LIN {X 0,Y 416.855,Z 989.857,A -85,B 0,C 180,E1 6681.651,E2 6681.651} C_VEL
LIN {X 0,Y 426.001,Z 970.369,A -85,B 0,C 180,E1 6680.53,E2 6680.53} C_VEL
LIN {X 0,Y 436.146,Z 946.367,A -85,B 0,C 180,E1 6679.376,E2 6679.376} C_VEL
LIN {X 0,Y 445.2,Z 921.165,A -85,B 0,C 180,E1 6678.399,E2 6678.399} C_VEL
LIN {X 0,Y 451.671,Z 900.478,A -85,B 0,C 180,E1 6677.741,E2 6677.741} C_VEL
LIN {X 0,Y 457.353,Z 879.296,A -85,B 0,C 180,E1 6677.183,E2 6677.183} C_VEL
LIN {X 0,Y 462.4,Z 856.717,A -85,B 0,C 180,E1 6676.706,E2 6676.706} C_VEL
LIN {X 0,Y 467.347,Z 827.03,A -85,B 0,C 180,E1 6676.196,E2 6676.196} C_VEL
LIN {X 0,Y 472.981,Z 773.128,A -85,B 0,C 180,E1 6675.392,E2 6675.392} C_VEL
LIN {X 0,Y 490.265,Z 601.502,A -85,B 0,C 180,E1 6672.888,E2 6672.888} C_VEL
LIN {X 0,Y 487.784,Z 596.947,A -85,B 0,C 180,E1 6670.631,E2 6670.631} C_VEL
LIN {X 0,Y 485.782,Z 593.042,A -85,B 0,C 180,E1 6668.101,E2 6668.101} C_VEL
LIN {X 0,Y 484.292,Z 588.607,A -85,B 0,C 180,E1 6662.84,E2 6662.84} C_VEL
LIN {X 0,Y 486.143,Z 593.645,A -85,B 0,C 180,E1 6657.171,E2 6657.171} C_VEL
LIN {X 0,Y 488.529,Z 598.315,A -85,B 0,C 180,E1 6654.421,E2 6654.421} C_VEL
LIN {X 0,Y 490.215,Z 601.519,A -85,B 0,C 180,E1 6652.939,E2 6652.939} C_VEL
LIN {X 0,Y 468.422,Z 816.947,A -85,B 0,C 180,E1 6649.795,E2 6649.795} C_VEL
LIN {X 0,Y 465.267,Z 839.316,A -85,B 0,C 180,E1 6649.432,E2 6649.432} C_VEL
LIN {X 0,Y 460.997,Z 861.82,A -85,B 0,C 180,E1 6649.009,E2 6649.009} C_VEL
LIN {X 0,Y 454.539,Z 888.776,A -85,B 0,C 180,E1 6648.359,E2 6648.359} C_VEL
LIN {X 0,Y 447.193,Z 913.264,A -85,B 0,C 180,E1 6647.605,E2 6647.605} C_VEL
LIN {X 0,Y 440.015,Z 933.977,A -85,B 0,C 180,E1 6646.83,E2 6646.83} C_VEL
LIN {X 0,Y 432.19,Z 953.973,A -85,B 0,C 180,E1 6645.941,E2 6645.941} C_VEL
LIN {X 0,Y 422.719,Z 975.589,A -85,B 0,C 180,E1 6644.807,E2 6644.807} C_VEL
LIN {X 0,Y 410.412,Z 1000.373,A -85,B 0,C 180,E1 6643.224,E2 6643.224} C_VEL
LIN {X 0,Y 400.027,Z 1019.259,A -85,B 0,C 180,E1 6641.769,E2 6641.769} C_VEL
LIN {X 0,Y 389.898,Z 1036.281,A -85,B 0,C 180,E1 6640.244,E2 6640.244} C_VEL
LIN {X 0,Y 379.202,Z 1053.022,A -85,B 0,C 180,E1 6638.499,E2 6638.499} C_VEL
LIN {X 0,Y 365.53,Z 1073.081,A -85,B 0,C 180,E1 6636.01,E2 6636.01} C_VEL
LIN {X 0,Y 351.999,Z 1091.305,A -85,B 0,C 180,E1 6633.222,E2 6633.222} C_VEL
LIN {X 0,Y 340.838,Z 1105.652,A -85,B 0,C 180,E1 6630.605,E2 6630.605} C_VEL
LIN {X 0,Y 329.999,Z 1119.088,A -85,B 0,C 180,E1 6627.708,E2 6627.708} C_VEL
LIN {X 0,Y 317.403,Z 1134.331,A -85,B 0,C 180,E1 6623.749,E2 6623.749} C_VEL
LIN {X 0,Y 306.251,Z 1147.367,A -85,B 0,C 180,E1 6619.526,E2 6619.526} C_VEL
LIN {X 0,Y 297.848,Z 1157.309,A -85,B 0,C 180,E1 6615.645,E2 6615.645} C_VEL
LIN {X 0,Y 290.31,Z 1166.501,A -85,B 0,C 180,E1 6611.336,E2 6611.336} C_VEL
LIN {X 0,Y 282.575,Z 1176.52,A -85,B 0,C 180,E1 6605.471,E2 6605.471} C_VEL
LIN {X 0,Y 278.125,Z 1182.904,A -85,B 0,C 180,E1 6600.696,E2 6600.696} C_VEL
LIN {X 0,Y 275.171,Z 1187.842,A -85,B 0,C 180,E1 6596.082,E2 6596.082} C_VEL
LIN {X 0,Y 273.379,Z 1191.521,A -85,B 0,C 180,E1 6591.678,E2 6591.678} C_VEL
LIN {X 0,Y 272.422,Z 1194.229,A -85,B 0,C 180,E1 6587.294,E2 6587.294} C_VEL
LIN {X 0,Y 272.031,Z 1195.927,A -85,B 0,C 180,E1 6583.172,E2 6583.172} C_VEL
LIN {X 0,Y 271.932,Z 1196.773,A -85,B 0,C 180,E1 6579.31,E2 6579.31} C_VEL
LIN {X 0,Y 271.908,Z 1196.87,A -85,B 0,C 180,E1 6575.274,E2 6575.274} C_VEL
LIN {X 0,Y 271.941,Z 1196.163,A -85,B 0,C 180,E1 6571.263,E2 6571.263} C_VEL
LIN {X 0,Y 272.119,Z 1194.546,A -85,B 0,C 180,E1 6567.05,E2 6567.05} C_VEL
LIN {X 0,Y 272.714,Z 1191.882,A -85,B 0,C 180,E1 6562.626,E2 6562.626} C_VEL
LIN {X 0,Y 273.987,Z 1188.224,A -85,B 0,C 180,E1 6558.207,E2 6558.207} C_VEL
LIN {X 0,Y 276.136,Z 1183.547,A -85,B 0,C 180,E1 6553.81,E2 6553.81} C_VEL
LIN {X 0,Y 279.466,Z 1177.53,A -85,B 0,C 180,E1 6549.255,E2 6549.255} C_VEL
LIN {X 0,Y 284.504,Z 1169.638,A -85,B 0,C 180,E1 6544.387,E2 6544.387} C_VEL
LIN {X 0,Y 291.973,Z 1158.86,A -85,B 0,C 180,E1 6539.09,E2 6539.09} C_VEL
LIN {X 0,Y 299.509,Z 1148.546,A -85,B 0,C 180,E1 6534.956,E2 6534.956} C_VEL
LIN {X 0,Y 307.424,Z 1137.911,A -85,B 0,C 180,E1 6531.356,E2 6531.356} C_VEL
LIN {X 0,Y 316.822,Z 1125.344,A -85,B 0,C 180,E1 6527.761,E2 6527.761} C_VEL
LIN {X 0,Y 329.366,Z 1108.186,A -85,B 0,C 180,E1 6523.737,E2 6523.737} C_VEL
LIN {X 0,Y 339.219,Z 1094.184,A -85,B 0,C 180,E1 6521.01,E2 6521.01} C_VEL
LIN {X 0,Y 349.142,Z 1079.549,A -85,B 0,C 180,E1 6518.572,E2 6518.572} C_VEL
LIN {X 0,Y 359.626,Z 1063.349,A -85,B 0,C 180,E1 6516.264,E2 6516.264} C_VEL
LIN {X 0,Y 372.238,Z 1042.639,A -85,B 0,C 180,E1 6513.782,E2 6513.782} C_VEL
LIN {X 0,Y 383.807,Z 1021.754,A -85,B 0,C 180,E1 6511.724,E2 6511.724} C_VEL
LIN {X 0,Y 393.285,Z 1003.316,A -85,B 0,C 180,E1 6510.184,E2 6510.184} C_VEL
LIN {X 0,Y 401.929,Z 985.07,A -85,B 0,C 180,E1 6508.875,E2 6508.875} C_VEL
LIN {X 0,Y 412.234,Z 961.113,A -85,B 0,C 180,E1 6507.409,E2 6507.409} C_VEL
LIN {X 0,Y 421.376,Z 936.508,A -85,B 0,C 180,E1 6506.191,E2 6506.191} C_VEL
LIN {X 0,Y 428.141,Z 915.89,A -85,B 0,C 180,E1 6505.338,E2 6505.338} C_VEL
LIN {X 0,Y 434.12,Z 895.023,A -85,B 0,C 180,E1 6504.612,E2 6504.612} C_VEL
LIN {X 0,Y 434.611,Z 893.203,A -85,B 0,C 180,E1 6504.555,E2 6504.555} C_VEL
LIN {X 0,Y 436.165,Z 886.037,A -85,B 0,C 180,E1 6504.214,E2 6504.214} C_VEL
LIN {X 0,Y 438.207,Z 868.294,A -85,B 0,C 180,E1 6502.999,E2 6502.999} C_VEL
LIN {X 0,Y 439.312,Z 860.964,A -85,B 0,C 180,E1 6502.707,E2 6502.707} C_VEL
LIN {X 0,Y 443.317,Z 838.651,A -85,B 0,C 180,E1 6502.264,E2 6502.264} C_VEL
LIN {X 0,Y 446.283,Z 816.191,A -85,B 0,C 180,E1 6501.884,E2 6501.884} C_VEL
LIN {X 0,Y 466.557,Z 598.28,A -85,B 0,C 180,E1 6498.618,E2 6498.618} C_VEL
LIN {X 0,Y 467.039,Z 592.534,A -85,B 0,C 180,E1 6498.505,E2 6498.505} C_VEL
LIN {X 0,Y 462.723,Z 584.65,A -85,B 0,C 180,E1 6495.864,E2 6495.864} C_VEL
LIN {X 0,Y 459.733,Z 579.467,A -85,B 0,C 180,E1 6493.65,E2 6493.65} C_VEL
LIN {X 0,Y 457.995,Z 576.374,A -85,B 0,C 180,E1 6492.098,E2 6492.098} C_VEL
LIN {X 0,Y 455.895,Z 572.558,A -85,B 0,C 180,E1 6489.723,E2 6489.723} C_VEL
LIN {X 0,Y 453.963,Z 568.532,A -85,B 0,C 180,E1 6486.069,E2 6486.069} C_VEL
LIN {X 0,Y 453.614,Z 568.037,A -85,B 0,C 180,E1 6484.805,E2 6484.805} C_VEL
LIN {X 0,Y 453.911,Z 568.255,A -85,B 0,C 180,E1 6480.252,E2 6480.252} C_VEL
LIN {X 0,Y 455.529,Z 572.159,A -85,B 0,C 180,E1 6476.854,E2 6476.854} C_VEL
LIN {X 0,Y 456.46,Z 573.573,A -85,B 0,C 180,E1 6475.666,E2 6475.666} C_VEL
LIN {X 0,Y 459.168,Z 578.446,A -85,B 0,C 180,E1 6472.933,E2 6472.933} C_VEL
LIN {X 0,Y 461.582,Z 582.786,A -85,B 0,C 180,E1 6471.027,E2 6471.027} C_VEL
LIN {X 0,Y 465.2,Z 589.229,A -85,B 0,C 180,E1 6468.658,E2 6468.658} C_VEL
LIN {X 0,Y 467.122,Z 592.997,A -85,B 0,C 180,E1 6467.535,E2 6467.535} C_VEL
LIN {X 0,Y 446.738,Z 813.471,A -85,B 0,C 180,E1 6464.235,E2 6464.235} C_VEL
LIN {X 0,Y 443.482,Z 839.489,A -85,B 0,C 180,E1 6463.8,E2 6463.8} C_VEL
LIN {X 0,Y 439.573,Z 861.723,A -85,B 0,C 180,E1 6463.373,E2 6463.373} C_VEL
LIN {X 0,Y 434.754,Z 883.632,A -85,B 0,C 180,E1 6462.854,E2 6462.854} C_VEL
LIN {X 0,Y 427.738,Z 910.07,A -85,B 0,C 180,E1 6462.065,E2 6462.065} C_VEL
LIN {X 0,Y 419.555,Z 935.282,A -85,B 0,C 180,E1 6461.108,E2 6461.108} C_VEL
LIN {X 0,Y 412.311,Z 954.975,A -85,B 0,C 180,E1 6460.208,E2 6460.208} C_VEL
LIN {X 0,Y 404.389,Z 974.343,A -85,B 0,C 180,E1 6459.169,E2 6459.169} C_VEL
LIN {X 0,Y 395.523,Z 994.037,A -85,B 0,C 180,E1 6457.928,E2 6457.928} C_VEL
LIN {X 0,Y 383.724,Z 1017.725,A -85,B 0,C 180,E1 6456.151,E2 6456.151} C_VEL
LIN {X 0,Y 372.705,Z 1037.638,A -85,B 0,C 180,E1 6454.345,E2 6454.345} C_VEL
LIN {X 0,Y 362.414,Z 1054.953,A -85,B 0,C 180,E1 6452.499,E2 6452.499} C_VEL
LIN {X 0,Y 351.852,Z 1071.672,A -85,B 0,C 180,E1 6450.41,E2 6450.41} C_VEL
LIN {X 0,Y 338.858,Z 1091.127,A -85,B 0,C 180,E1 6447.518,E2 6447.518} C_VEL
LIN {X 0,Y 326.855,Z 1107.895,A -85,B 0,C 180,E1 6444.462,E2 6444.462} C_VEL
LIN {X 0,Y 316.79,Z 1121.525,A -85,B 0,C 180,E1 6441.514,E2 6441.514} C_VEL
LIN {X 0,Y 307.034,Z 1134.431,A -85,B 0,C 180,E1 6438.225,E2 6438.225} C_VEL
LIN {X 0,Y 296.536,Z 1148.302,A -85,B 0,C 180,E1 6433.996,E2 6433.996} C_VEL
LIN {X 0,Y 287.11,Z 1160.609,A -85,B 0,C 180,E1 6429.334,E2 6429.334} C_VEL
LIN {X 0,Y 280.577,Z 1169.55,A -85,B 0,C 180,E1 6425.262,E2 6425.262} C_VEL
LIN {X 0,Y 275.039,Z 1177.571,A -85,B 0,C 180,E1 6420.91,E2 6420.91} C_VEL
LIN {X 0,Y 270.647,Z 1184.594,A -85,B 0,C 180,E1 6416.317,E2 6416.317} C_VEL
LIN {X 0,Y 266.919,Z 1191.693,A -85,B 0,C 180,E1 6410.525,E2 6410.525} C_VEL
LIN {X 0,Y 264.96,Z 1196.582,A -85,B 0,C 180,E1 6405.094,E2 6405.094} C_VEL
LIN {X 0,Y 264.183,Z 1199.646,A -85,B 0,C 180,E1 6400.468,E2 6400.468} C_VEL
LIN {X 0,Y 263.954,Z 1201.529,A -85,B 0,C 180,E1 6396.308,E2 6396.308} C_VEL
LIN {X 0,Y 263.915,Z 1202.571,A -85,B 0,C 180,E1 6392.172,E2 6392.172} C_VEL
LIN {X 0,Y 263.913,Z 1202.76,A -85,B 0,C 180,E1 6387.83,E2 6387.83} C_VEL
LIN {X 0,Y 263.958,Z 1202.033,A -85,B 0,C 180,E1 6383.476,E2 6383.476} C_VEL
LIN {X 0,Y 264.264,Z 1200.282,A -85,B 0,C 180,E1 6378.875,E2 6378.875} C_VEL
LIN {X 0,Y 265.179,Z 1197.53,A -85,B 0,C 180,E1 6374.248,E2 6374.248} C_VEL
LIN {X 0,Y 266.953,Z 1193.765,A -85,B 0,C 180,E1 6369.616,E2 6369.616} C_VEL
LIN {X 0,Y 269.817,Z 1188.967,A -85,B 0,C 180,E1 6365.011,E2 6365.011} C_VEL
LIN {X 0,Y 274.125,Z 1182.778,A -85,B 0,C 180,E1 6360.242,E2 6360.242} C_VEL
LIN {X 0,Y 280.711,Z 1174.386,A -85,B 0,C 180,E1 6355.008,E2 6355.008} C_VEL
LIN {X 0,Y 289.919,Z 1163.295,A -85,B 0,C 180,E1 6349.582,E2 6349.582} C_VEL
LIN {X 0,Y 298.594,Z 1153.259,A -85,B 0,C 180,E1 6345.585,E2 6345.585} C_VEL
LIN {X 0,Y 308.005,Z 1142.435,A -85,B 0,C 180,E1 6341.971,E2 6341.971} C_VEL
LIN {X 0,Y 319.554,Z 1129.067,A -85,B 0,C 180,E1 6338.246,E2 6338.246} C_VEL
LIN {X 0,Y 333.497,Z 1112.298,A -85,B 0,C 180,E1 6334.464,E2 6334.464} C_VEL
LIN {X 0,Y 345.466,Z 1097.29,A -85,B 0,C 180,E1 6331.69,E2 6331.69} C_VEL
LIN {X 0,Y 356.816,Z 1082.405,A -85,B 0,C 180,E1 6329.367,E2 6329.367} C_VEL
LIN {X 0,Y 369.062,Z 1065.458,A -85,B 0,C 180,E1 6327.13,E2 6327.13} C_VEL
LIN {X 0,Y 384.064,Z 1042.943,A -85,B 0,C 180,E1 6324.691,E2 6324.691} C_VEL
LIN {X 0,Y 394.923,Z 1025.236,A -85,B 0,C 180,E1 6323.106,E2 6323.106} C_VEL
LIN {X 0,Y 405.046,Z 1007.376,A -85,B 0,C 180,E1 6321.733,E2 6321.733} C_VEL
LIN {X 0,Y 414.747,Z 988.785,A -85,B 0,C 180,E1 6320.514,E2 6320.514} C_VEL
LIN {X 0,Y 424.44,Z 968.395,A -85,B 0,C 180,E1 6319.378,E2 6319.378} C_VEL
LIN {X 0,Y 435.63,Z 941.619,A -85,B 0,C 180,E1 6318.155,E2 6318.155} C_VEL
LIN {X 0,Y 443.597,Z 919.527,A -85,B 0,C 180,E1 6317.338,E2 6317.338} C_VEL
LIN {X 0,Y 449.955,Z 899.331,A -85,B 0,C 180,E1 6316.716,E2 6316.716} C_VEL
LIN {X 0,Y 455.67,Z 878.172,A -85,B 0,C 180,E1 6316.176,E2 6316.176} C_VEL
LIN {X 0,Y 461.272,Z 853.11,A -85,B 0,C 180,E1 6315.67,E2 6315.67} C_VEL
LIN {X 0,Y 465.812,Z 824.74,A -85,B 0,C 180,E1 6315.2,E2 6315.2} C_VEL
LIN {X 0,Y 473.898,Z 747.238,A -85,B 0,C 180,E1 6314.062,E2 6314.062} C_VEL
LIN {X 0,Y 488.256,Z 607.87,A -85,B 0,C 180,E1 6312.057,E2 6312.057} C_VEL
LIN {X 0,Y 486.579,Z 604.671,A -85,B 0,C 180,E1 6310.418,E2 6310.418} C_VEL
LIN {X 0,Y 484.772,Z 600.976,A -85,B 0,C 180,E1 6308.063,E2 6308.063} C_VEL
LIN {X 0,Y 483.312,Z 596.579,A -85,B 0,C 180,E1 6302.846,E2 6302.846} C_VEL
LIN {X 0,Y 485.071,Z 601.541,A -85,B 0,C 180,E1 6297.283,E2 6297.283} C_VEL
LIN {X 0,Y 487.35,Z 606.118,A -85,B 0,C 180,E1 6294.584,E2 6294.584} C_VEL
LIN {X 0,Y 488.188,Z 608.003,A -85,B 0,C 180,E1 6293.774,E2 6293.774} C_VEL
LIN {X 0,Y 466.314,Z 819.614,A -85,B 0,C 180,E1 6290.714,E2 6290.714} C_VEL
LIN {X 0,Y 462.847,Z 842.858,A -85,B 0,C 180,E1 6290.338,E2 6290.338} C_VEL
LIN {X 0,Y 456.918,Z 871.614,A -85,B 0,C 180,E1 6289.772,E2 6289.772} C_VEL
LIN {X 0,Y 450.694,Z 895.154,A -85,B 0,C 180,E1 6289.169,E2 6289.169} C_VEL
LIN {X 0,Y 444.315,Z 915.662,A -85,B 0,C 180,E1 6288.53,E2 6288.53} C_VEL
LIN {X 0,Y 437.322,Z 935.333,A -85,B 0,C 180,E1 6287.798,E2 6287.798} C_VEL
LIN {X 0,Y 429.119,Z 955.802,A -85,B 0,C 180,E1 6286.895,E2 6286.895} C_VEL
LIN {X 0,Y 417.977,Z 980.398,A -85,B 0,C 180,E1 6285.594,E2 6285.594} C_VEL
LIN {X 0,Y 406.456,Z 1002.68,A -85,B 0,C 180,E1 6284.153,E2 6284.153} C_VEL
LIN {X 0,Y 396.249,Z 1020.763,A -85,B 0,C 180,E1 6282.761,E2 6282.761} C_VEL
LIN {X 0,Y 386,Z 1037.532,A -85,B 0,C 180,E1 6281.264,E2 6281.264} C_VEL
LIN {X 0,Y 373.867,Z 1056.004,A -85,B 0,C 180,E1 6279.327,E2 6279.327} C_VEL
LIN {X 0,Y 359.225,Z 1076.511,A -85,B 0,C 180,E1 6276.71,E2 6276.71} C_VEL
LIN {X 0,Y 347.305,Z 1092.092,A -85,B 0,C 180,E1 6274.303,E2 6274.303} C_VEL
LIN {X 0,Y 336.022,Z 1106.146,A -85,B 0,C 180,E1 6271.735,E2 6271.735} C_VEL
LIN {X 0,Y 324.838,Z 1119.541,A -85,B 0,C 180,E1 6268.836,E2 6268.836} C_VEL
LIN {X 0,Y 311.789,Z 1134.715,A -85,B 0,C 180,E1 6264.86,E2 6264.86} C_VEL
LIN {X 0,Y 300.671,Z 1147.194,A -85,B 0,C 180,E1 6260.789,E2 6260.789} C_VEL
LIN {X 0,Y 291.825,Z 1157.164,A -85,B 0,C 180,E1 6256.868,E2 6256.868} C_VEL
LIN {X 0,Y 284.076,Z 1166.104,A -85,B 0,C 180,E1 6252.639,E2 6252.639} C_VEL
LIN {X 0,Y 276.368,Z 1175.533,A -85,B 0,C 180,E1 6247.17,E2 6247.17} C_VEL
LIN {X 0,Y 270.789,Z 1182.864,A -85,B 0,C 180,E1 6241.622,E2 6241.622} C_VEL
LIN {X 0,Y 267.559,Z 1187.826,A -85,B 0,C 180,E1 6236.883,E2 6236.883} C_VEL
LIN {X 0,Y 265.582,Z 1191.529,A -85,B 0,C 180,E1 6232.348,E2 6232.348} C_VEL
LIN {X 0,Y 264.503,Z 1194.261,A -85,B 0,C 180,E1 6227.829,E2 6227.829} C_VEL
LIN {X 0,Y 264.055,Z 1195.982,A -85,B 0,C 180,E1 6223.577,E2 6223.577} C_VEL
LIN {X 0,Y 263.934,Z 1196.85,A -85,B 0,C 180,E1 6219.594,E2 6219.594} C_VEL
LIN {X 0,Y 263.909,Z 1196.969,A -85,B 0,C 180,E1 6215.434,E2 6215.434} C_VEL
LIN {X 0,Y 263.941,Z 1196.285,A -85,B 0,C 180,E1 6211.302,E2 6211.302} C_VEL
LIN {X 0,Y 264.144,Z 1194.579,A -85,B 0,C 180,E1 6206.744,E2 6206.744} C_VEL
LIN {X 0,Y 264.803,Z 1191.893,A -85,B 0,C 180,E1 6202.187,E2 6202.187} C_VEL
LIN {X 0,Y 266.209,Z 1188.155,A -85,B 0,C 180,E1 6197.574,E2 6197.574} C_VEL
LIN {X 0,Y 268.513,Z 1183.515,A -85,B 0,C 180,E1 6193.114,E2 6193.114} C_VEL
LIN {X 0,Y 271.894,Z 1177.77,A -85,B 0,C 180,E1 6188.649,E2 6188.649} C_VEL
LIN {X 0,Y 276.938,Z 1170.247,A -85,B 0,C 180,E1 6183.865,E2 6183.865} C_VEL
LIN {X 0,Y 285.017,Z 1159.177,A -85,B 0,C 180,E1 6178.249,E2 6178.249} C_VEL
LIN {X 0,Y 292.974,Z 1148.744,A -85,B 0,C 180,E1 6173.985,E2 6173.985} C_VEL
LIN {X 0,Y 301.094,Z 1138.281,A -85,B 0,C 180,E1 6170.386,E2 6170.386} C_VEL
LIN {X 0,Y 310.348,Z 1126.364,A -85,B 0,C 180,E1 6166.919,E2 6166.919} C_VEL
LIN {X 0,Y 323.031,Z 1109.711,A -85,B 0,C 180,E1 6162.92,E2 6162.92} C_VEL
LIN {X 0,Y 333.957,Z 1094.677,A -85,B 0,C 180,E1 6159.961,E2 6159.961} C_VEL
LIN {X 0,Y 344.155,Z 1080.078,A -85,B 0,C 180,E1 6157.519,E2 6157.519} C_VEL
LIN {X 0,Y 354.584,Z 1064.41,A -85,B 0,C 180,E1 6155.278,E2 6155.278} C_VEL
LIN {X 0,Y 366.856,Z 1044.878,A -85,B 0,C 180,E1 6152.916,E2 6152.916} C_VEL
LIN {X 0,Y 379.299,Z 1023.117,A -85,B 0,C 180,E1 6150.753,E2 6150.753} C_VEL
LIN {X 0,Y 388.761,Z 1005.204,A -85,B 0,C 180,E1 6149.254,E2 6149.254} C_VEL
LIN {X 0,Y 397.394,Z 987.488,A -85,B 0,C 180,E1 6147.975,E2 6147.975} C_VEL
LIN {X 0,Y 405.934,Z 968.287,A -85,B 0,C 180,E1 6146.776,E2 6146.776} C_VEL
LIN {X 0,Y 415.123,Z 945.419,A -85,B 0,C 180,E1 6145.573,E2 6145.573} C_VEL
LIN {X 0,Y 424.04,Z 919.652,A -85,B 0,C 180,E1 6144.469,E2 6144.469} C_VEL
LIN {X 0,Y 430.538,Z 897.744,A -85,B 0,C 180,E1 6143.7,E2 6143.7} C_VEL
LIN {X 0,Y 435.93,Z 876.487,A -85,B 0,C 180,E1 6143.083,E2 6143.083} C_VEL
LIN {X 0,Y 439.312,Z 860.964,A -85,B 0,C 180,E1 6142.707,E2 6142.707} C_VEL
LIN {X 0,Y 440.435,Z 853.582,A -85,B 0,C 180,E1 6142.424,E2 6142.424} C_VEL
LIN {X 0,Y 441.852,Z 834.293,A -85,B 0,C 180,E1 6141.283,E2 6141.283} C_VEL
LIN {X 0,Y 442.463,Z 827.846,A -85,B 0,C 180,E1 6141.087,E2 6141.087} C_VEL
LIN {X 0,Y 447.025,Z 782.963,A -85,B 0,C 180,E1 6140.397,E2 6140.397} C_VEL
LIN {X 0,Y 464.486,Z 598.22,A -85,B 0,C 180,E1 6137.654,E2 6137.654} C_VEL
LIN {X 0,Y 460.671,Z 591.177,A -85,B 0,C 180,E1 6135.162,E2 6135.162} C_VEL
LIN {X 0,Y 458.162,Z 586.637,A -85,B 0,C 180,E1 6133.183,E2 6133.183} C_VEL
LIN {X 0,Y 456.632,Z 583.895,A -85,B 0,C 180,E1 6131.75,E2 6131.75} C_VEL
LIN {X 0,Y 454.824,Z 580.443,A -85,B 0,C 180,E1 6129.618,E2 6129.618} C_VEL
LIN {X 0,Y 452.946,Z 576.425,A -85,B 0,C 180,E1 6125.955,E2 6125.955} C_VEL
LIN {X 0,Y 452.565,Z 575.934,A -85,B 0,C 180,E1 6124.435,E2 6124.435} C_VEL
LIN {X 0,Y 452.919,Z 576.315,A -85,B 0,C 180,E1 6120.253,E2 6120.253} C_VEL
LIN {X 0,Y 454.733,Z 580.388,A -85,B 0,C 180,E1 6116.596,E2 6116.596} C_VEL
LIN {X 0,Y 455.558,Z 581.953,A -85,B 0,C 180,E1 6115.531,E2 6115.531} C_VEL
LIN {X 0,Y 457.887,Z 586.121,A -85,B 0,C 180,E1 6113.165,E2 6113.165} C_VEL
LIN {X 0,Y 460.24,Z 590.471,A -85,B 0,C 180,E1 6111.253,E2 6111.253} C_VEL
LIN {X 0,Y 463.779,Z 596.967,A -85,B 0,C 180,E1 6108.874,E2 6108.874} C_VEL
LIN {X 0,Y 464.522,Z 598.688,A -85,B 0,C 180,E1 6108.405,E2 6108.405} C_VEL
LIN {X 0,Y 443.835,Z 817.103,A -85,B 0,C 180,E1 6105.158,E2 6105.158} C_VEL
LIN {X 0,Y 440.777,Z 840.468,A -85,B 0,C 180,E1 6104.768,E2 6104.768} C_VEL
LIN {X 0,Y 436.776,Z 862.653,A -85,B 0,C 180,E1 6104.346,E2 6104.346} C_VEL
LIN {X 0,Y 431.448,Z 886.228,A -85,B 0,C 180,E1 6103.79,E2 6103.79} C_VEL
LIN {X 0,Y 423.603,Z 914.226,A -85,B 0,C 180,E1 6102.935,E2 6102.935} C_VEL
LIN {X 0,Y 416.546,Z 935.471,A -85,B 0,C 180,E1 6102.131,E2 6102.131} C_VEL
LIN {X 0,Y 408.996,Z 955.598,A -85,B 0,C 180,E1 6101.223,E2 6101.223} C_VEL
LIN {X 0,Y 400.625,Z 975.615,A -85,B 0,C 180,E1 6100.158,E2 6100.158} C_VEL
LIN {X 0,Y 389.678,Z 999.236,A -85,B 0,C 180,E1 6098.659,E2 6098.659} C_VEL
LIN {X 0,Y 378.143,Z 1021.212,A -85,B 0,C 180,E1 6096.953,E2 6096.953} C_VEL
LIN {X 0,Y 368.167,Z 1038.749,A -85,B 0,C 180,E1 6095.35,E2 6095.35} C_VEL
LIN {X 0,Y 357.904,Z 1055.574,A -85,B 0,C 180,E1 6093.558,E2 6093.558} C_VEL
LIN {X 0,Y 346.69,Z 1072.843,A -85,B 0,C 180,E1 6091.395,E2 6091.395} C_VEL
LIN {X 0,Y 332.11,Z 1093.801,A -85,B 0,C 180,E1 6088.205,E2 6088.205} C_VEL
LIN {X 0,Y 320.819,Z 1109.09,A -85,B 0,C 180,E1 6085.366,E2 6085.366} C_VEL
LIN {X 0,Y 310.486,Z 1122.603,A -85,B 0,C 180,E1 6082.393,E2 6082.393} C_VEL
LIN {X 0,Y 299.954,Z 1136.051,A -85,B 0,C 180,E1 6078.883,E2 6078.883} C_VEL
LIN {X 0,Y 287.97,Z 1151.074,A -85,B 0,C 180,E1 6074.049,E2 6074.049} C_VEL
LIN {X 0,Y 279.886,Z 1161.288,A -85,B 0,C 180,E1 6070.02,E2 6070.02} C_VEL
LIN {X 0,Y 273.124,Z 1170.142,A -85,B 0,C 180,E1 6065.856,E2 6065.856} C_VEL
LIN {X 0,Y 267.312,Z 1178.185,A -85,B 0,C 180,E1 6061.328,E2 6061.328} C_VEL
LIN {X 0,Y 261.961,Z 1186.53,A -85,B 0,C 180,E1 6055.551,E2 6055.551} C_VEL
LIN {X 0,Y 258.589,Z 1192.715,A -85,B 0,C 180,E1 6049.894,E2 6049.894} C_VEL
LIN {X 0,Y 256.954,Z 1196.766,A -85,B 0,C 180,E1 6045.113,E2 6045.113} C_VEL
LIN {X 0,Y 256.19,Z 1199.635,A -85,B 0,C 180,E1 6040.571,E2 6040.571} C_VEL
LIN {X 0,Y 255.953,Z 1201.488,A -85,B 0,C 180,E1 6036.281,E2 6036.281} C_VEL
LIN {X 0,Y 255.915,Z 1202.499,A -85,B 0,C 180,E1 6032.016,E2 6032.016} C_VEL
LIN {X 0,Y 255.913,Z 1202.679,A -85,B 0,C 180,E1 6027.762,E2 6027.762} C_VEL
LIN {X 0,Y 255.963,Z 1201.967,A -85,B 0,C 180,E1 6023.271,E2 6023.271} C_VEL
LIN {X 0,Y 256.302,Z 1200.231,A -85,B 0,C 180,E1 6018.525,E2 6018.525} C_VEL
LIN {X 0,Y 257.326,Z 1197.452,A -85,B 0,C 180,E1 6013.693,E2 6013.693} C_VEL
LIN {X 0,Y 259.35,Z 1193.539,A -85,B 0,C 180,E1 6008.753,E2 6008.753} C_VEL
LIN {X 0,Y 262.494,Z 1188.709,A -85,B 0,C 180,E1 6004.021,E2 6004.021} C_VEL
LIN {X 0,Y 267.137,Z 1182.515,A -85,B 0,C 180,E1 5999.152,E2 5999.152} C_VEL
LIN {X 0,Y 274.542,Z 1173.717,A -85,B 0,C 180,E1 5993.585,E2 5993.585} C_VEL
LIN {X 0,Y 284.028,Z 1162.882,A -85,B 0,C 180,E1 5988.273,E2 5988.273} C_VEL
LIN {X 0,Y 292.666,Z 1153.357,A -85,B 0,C 180,E1 5984.437,E2 5984.437} C_VEL
LIN {X 0,Y 302.444,Z 1142.572,A -85,B 0,C 180,E1 5980.795,E2 5980.795} C_VEL
LIN {X 0,Y 313.871,Z 1129.843,A -85,B 0,C 180,E1 5977.213,E2 5977.213} C_VEL
LIN {X 0,Y 328.859,Z 1112.496,A -85,B 0,C 180,E1 5973.269,E2 5973.269} C_VEL
LIN {X 0,Y 341.184,Z 1097.521,A -85,B 0,C 180,E1 5970.505,E2 5970.505} C_VEL
LIN {X 0,Y 352.831,Z 1082.673,A -85,B 0,C 180,E1 5968.198,E2 5968.198} C_VEL
LIN {X 0,Y 365.017,Z 1066.252,A -85,B 0,C 180,E1 5966.043,E2 5966.043} C_VEL
LIN {X 0,Y 379.964,Z 1044.518,A -85,B 0,C 180,E1 5963.688,E2 5963.688} C_VEL
LIN {X 0,Y 392.109,Z 1025.138,A -85,B 0,C 180,E1 5961.97,E2 5961.97} C_VEL
LIN {X 0,Y 402.277,Z 1007.566,A -85,B 0,C 180,E1 5960.643,E2 5960.643} C_VEL
LIN {X 0,Y 412.4,Z 988.52,A -85,B 0,C 180,E1 5959.416,E2 5959.416} C_VEL
LIN {X 0,Y 422.721,Z 967.135,A -85,B 0,C 180,E1 5958.256,E2 5958.256} C_VEL
LIN {X 0,Y 433.631,Z 941.281,A -85,B 0,C 180,E1 5957.108,E2 5957.108} C_VEL
LIN {X 0,Y 441.292,Z 920.418,A -85,B 0,C 180,E1 5956.352,E2 5956.352} C_VEL
LIN {X 0,Y 447.952,Z 899.648,A -85,B 0,C 180,E1 5955.723,E2 5955.723} C_VEL
LIN {X 0,Y 453.8,Z 878.354,A -85,B 0,C 180,E1 5955.192,E2 5955.192} C_VEL
LIN {X 0,Y 459.311,Z 854.109,A -85,B 0,C 180,E1 5954.712,E2 5954.712} C_VEL
LIN {X 0,Y 464.11,Z 824.968,A -85,B 0,C 180,E1 5954.235,E2 5954.235} C_VEL
LIN {X 0,Y 471.725,Z 753.59,A -85,B 0,C 180,E1 5953.198,E2 5953.198} C_VEL
LIN {X 0,Y 486.332,Z 614.23,A -85,B 0,C 180,E1 5951.203,E2 5951.203} C_VEL
LIN {X 0,Y 484.867,Z 611.502,A -85,B 0,C 180,E1 5949.616,E2 5949.616} C_VEL
LIN {X 0,Y 483.641,Z 608.779,A -85,B 0,C 180,E1 5947.843,E2 5947.843} C_VEL
LIN {X 0,Y 482.32,Z 604.661,A -85,B 0,C 180,E1 5942.733,E2 5942.733} C_VEL
LIN {X 0,Y 484,Z 609.437,A -85,B 0,C 180,E1 5937.395,E2 5937.395} C_VEL
LIN {X 0,Y 486.175,Z 613.92,A -85,B 0,C 180,E1 5934.749,E2 5934.749} C_VEL
LIN {X 0,Y 486.28,Z 614.379,A -85,B 0,C 180,E1 5934.618,E2 5934.618} C_VEL
LIN {X 0,Y 464.53,Z 820.666,A -85,B 0,C 180,E1 5931.666,E2 5931.666} C_VEL
LIN {X 0,Y 460.616,Z 846.004,A -85,B 0,C 180,E1 5931.26,E2 5931.26} C_VEL
LIN {X 0,Y 454.561,Z 873.901,A -85,B 0,C 180,E1 5930.707,E2 5930.707} C_VEL
LIN {X 0,Y 448.785,Z 895.326,A -85,B 0,C 180,E1 5930.165,E2 5930.165} C_VEL
LIN {X 0,Y 442.293,Z 915.88,A -85,B 0,C 180,E1 5929.538,E2 5929.538} C_VEL
LIN {X 0,Y 435.197,Z 935.532,A -85,B 0,C 180,E1 5928.823,E2 5928.823} C_VEL
LIN {X 0,Y 426.43,Z 957.016,A -85,B 0,C 180,E1 5927.892,E2 5927.892} C_VEL
LIN {X 0,Y 414.347,Z 982.869,A -85,B 0,C 180,E1 5926.528,E2 5926.528} C_VEL
LIN {X 0,Y 403.508,Z 1003.375,A -85,B 0,C 180,E1 5925.212,E2 5925.212} C_VEL
LIN {X 0,Y 393.411,Z 1020.899,A -85,B 0,C 180,E1 5923.883,E2 5923.883} C_VEL
LIN {X 0,Y 382.535,Z 1038.308,A -85,B 0,C 180,E1 5922.35,E2 5922.35} C_VEL
LIN {X 0,Y 368.608,Z 1058.981,A -85,B 0,C 180,E1 5920.179,E2 5920.179} C_VEL
LIN {X 0,Y 354.437,Z 1078.042,A -85,B 0,C 180,E1 5917.711,E2 5917.711} C_VEL
LIN {X 0,Y 342.595,Z 1093.063,A -85,B 0,C 180,E1 5915.383,E2 5915.383} C_VEL
LIN {X 0,Y 330.683,Z 1107.426,A -85,B 0,C 180,E1 5912.741,E2 5912.741} C_VEL
LIN {X 0,Y 316.764,Z 1123.552,A -85,B 0,C 180,E1 5909.155,E2 5909.155} C_VEL
LIN {X 0,Y 304.091,Z 1137.439,A -85,B 0,C 180,E1 5905.286,E2 5905.286} C_VEL
LIN {X 0,Y 294.254,Z 1148.073,A -85,B 0,C 180,E1 5901.714,E2 5901.714} C_VEL
LIN {X 0,Y 285.512,Z 1157.487,A -85,B 0,C 180,E1 5897.938,E2 5897.938} C_VEL
LIN {X 0,Y 277.187,Z 1166.618,A -85,B 0,C 180,E1 5893.525,E2 5893.525} C_VEL
LIN {X 0,Y 268.614,Z 1176.478,A -85,B 0,C 180,E1 5887.545,E2 5887.545} C_VEL
LIN {X 0,Y 263.322,Z 1183.081,A -85,B 0,C 180,E1 5882.37,E2 5882.37} C_VEL
LIN {X 0,Y 259.859,Z 1188.019,A -85,B 0,C 180,E1 5877.498,E2 5877.498} C_VEL
LIN {X 0,Y 257.733,Z 1191.698,A -85,B 0,C 180,E1 5872.826,E2 5872.826} C_VEL
LIN {X 0,Y 256.556,Z 1194.406,A -85,B 0,C 180,E1 5868.166,E2 5868.166} C_VEL
LIN {X 0,Y 256.069,Z 1196.104,A -85,B 0,C 180,E1 5863.779,E2 5863.779} C_VEL
LIN {X 0,Y 255.935,Z 1196.949,A -85,B 0,C 180,E1 5859.67,E2 5859.67} C_VEL
LIN {X 0,Y 255.909,Z 1197.069,A -85,B 0,C 180,E1 5855.605,E2 5855.605} C_VEL
LIN {X 0,Y 255.944,Z 1196.339,A -85,B 0,C 180,E1 5851.118,E2 5851.118} C_VEL
LIN {X 0,Y 256.153,Z 1194.723,A -85,B 0,C 180,E1 5846.642,E2 5846.642} C_VEL
LIN {X 0,Y 256.853,Z 1192.061,A -85,B 0,C 180,E1 5841.943,E2 5841.943} C_VEL
LIN {X 0,Y 258.315,Z 1188.404,A -85,B 0,C 180,E1 5837.253,E2 5837.253} C_VEL
LIN {X 0,Y 260.783,Z 1183.73,A -85,B 0,C 180,E1 5832.598,E2 5832.598} C_VEL
LIN {X 0,Y 264.353,Z 1178.009,A -85,B 0,C 180,E1 5828.009,E2 5828.009} C_VEL
LIN {X 0,Y 269.396,Z 1170.857,A -85,B 0,C 180,E1 5823.313,E2 5823.313} C_VEL
LIN {X 0,Y 277.443,Z 1160.389,A -85,B 0,C 180,E1 5817.765,E2 5817.765} C_VEL
LIN {X 0,Y 286.298,Z 1149.229,A -85,B 0,C 180,E1 5813.079,E2 5813.079} C_VEL
LIN {X 0,Y 294.855,Z 1138.65,A -85,B 0,C 180,E1 5809.376,E2 5809.376} C_VEL
LIN {X 0,Y 304.448,Z 1126.758,A -85,B 0,C 180,E1 5805.872,E2 5805.872} C_VEL
LIN {X 0,Y 317.227,Z 1110.609,A -85,B 0,C 180,E1 5801.938,E2 5801.938} C_VEL
LIN {X 0,Y 329.414,Z 1094.341,A -85,B 0,C 180,E1 5798.731,E2 5798.731} C_VEL
LIN {X 0,Y 339.928,Z 1079.696,A -85,B 0,C 180,E1 5796.297,E2 5796.297} C_VEL
LIN {X 0,Y 350.983,Z 1063.486,A -85,B 0,C 180,E1 5794.003,E2 5794.003} C_VEL
LIN {X 0,Y 364.344,Z 1042.576,A -85,B 0,C 180,E1 5791.533,E2 5791.533} C_VEL
LIN {X 0,Y 376.341,Z 1021.859,A -85,B 0,C 180,E1 5789.527,E2 5789.527} C_VEL
LIN {X 0,Y 386.224,Z 1003.404,A -85,B 0,C 180,E1 5788.017,E2 5788.017} C_VEL
LIN {X 0,Y 395.23,Z 985.139,A -85,B 0,C 180,E1 5786.741,E2 5786.741} C_VEL
LIN {X 0,Y 405.602,Z 961.917,A -85,B 0,C 180,E1 5785.354,E2 5785.354} C_VEL
LIN {X 0,Y 415.289,Z 936.857,A -85,B 0,C 180,E1 5784.145,E2 5784.145} C_VEL
LIN {X 0,Y 422.408,Z 915.858,A -85,B 0,C 180,E1 5783.302,E2 5783.302} C_VEL
LIN {X 0,Y 428.597,Z 894.923,A -85,B 0,C 180,E1 5782.6,E2 5782.6} C_VEL
LIN {X 0,Y 434.571,Z 871.147,A -85,B 0,C 180,E1 5781.947,E2 5781.947} C_VEL
LIN {X 0,Y 440.176,Z 842.487,A -85,B 0,C 180,E1 5781.345,E2 5781.345} C_VEL
LIN {X 0,Y 442.463,Z 827.846,A -85,B 0,C 180,E1 5781.087,E2 5781.087} C_VEL
LIN {X 0,Y 443.043,Z 820.326,A -85,B 0,C 180,E1 5780.847,E2 5780.847} C_VEL
LIN {X 0,Y 443.261,Z 800.783,A -85,B 0,C 180,E1 5779.766,E2 5779.766} C_VEL
LIN {X 0,Y 443.655,Z 794.3,A -85,B 0,C 180,E1 5779.576,E2 5779.576} C_VEL
LIN {X 0,Y 462.005,Z 603.818,A -85,B 0,C 180,E1 5776.771,E2 5776.771} C_VEL
LIN {X 0,Y 458.002,Z 596.246,A -85,B 0,C 180,E1 5773.895,E2 5773.895} C_VEL
LIN {X 0,Y 455.53,Z 591.801,A -85,B 0,C 180,E1 5771.651,E2 5771.651} C_VEL
LIN {X 0,Y 453.755,Z 588.328,A -85,B 0,C 180,E1 5769.513,E2 5769.513} C_VEL
LIN {X 0,Y 451.796,Z 583.984,A -85,B 0,C 180,E1 5765.334,E2 5765.334} C_VEL
LIN {X 0,Y 451.877,Z 584.028,A -85,B 0,C 180,E1 5760.507,E2 5760.507} C_VEL
LIN {X 0,Y 453.563,Z 588.142,A -85,B 0,C 180,E1 5756.841,E2 5756.841} C_VEL
LIN {X 0,Y 454.362,Z 589.632,A -85,B 0,C 180,E1 5755.772,E2 5755.772} C_VEL
LIN {X 0,Y 456.679,Z 593.932,A -85,B 0,C 180,E1 5753.336,E2 5753.336} C_VEL
LIN {X 0,Y 458.906,Z 598.154,A -85,B 0,C 180,E1 5751.48,E2 5751.48} C_VEL
LIN {X 0,Y 462.046,Z 604.17,A -85,B 0,C 180,E1 5749.288,E2 5749.288} C_VEL
LIN {X 0,Y 441.23,Z 819.116,A -85,B 0,C 180,E1 5746.119,E2 5746.119} C_VEL
LIN {X 0,Y 438.196,Z 841.451,A -85,B 0,C 180,E1 5745.748,E2 5745.748} C_VEL
LIN {X 0,Y 434.015,Z 864.023,A -85,B 0,C 180,E1 5745.322,E2 5745.322} C_VEL
LIN {X 0,Y 427.709,Z 890.935,A -85,B 0,C 180,E1 5744.682,E2 5744.682} C_VEL
LIN {X 0,Y 420.415,Z 915.761,A -85,B 0,C 180,E1 5743.913,E2 5743.913} C_VEL
LIN {X 0,Y 413.673,Z 935.657,A -85,B 0,C 180,E1 5743.169,E2 5743.169} C_VEL
LIN {X 0,Y 406.184,Z 955.29,A -85,B 0,C 180,E1 5742.3,E2 5742.3} C_VEL
LIN {X 0,Y 397.982,Z 974.609,A -85,B 0,C 180,E1 5741.293,E2 5741.293} C_VEL
LIN {X 0,Y 388.322,Z 995.222,A -85,B 0,C 180,E1 5740.023,E2 5740.023} C_VEL
LIN {X 0,Y 375.73,Z 1019.243,A -85,B 0,C 180,E1 5738.241,E2 5738.241} C_VEL
LIN {X 0,Y 364.635,Z 1038.383,A -85,B 0,C 180,E1 5736.527,E2 5736.527} C_VEL
LIN {X 0,Y 353.883,Z 1055.62,A -85,B 0,C 180,E1 5734.709,E2 5734.709} C_VEL
LIN {X 0,Y 342.458,Z 1072.787,A -85,B 0,C 180,E1 5732.573,E2 5732.573} C_VEL
LIN {X 0,Y 327.541,Z 1093.651,A -85,B 0,C 180,E1 5729.414,E2 5729.414} C_VEL
LIN {X 0,Y 315.923,Z 1108.916,A -85,B 0,C 180,E1 5726.584,E2 5726.584} C_VEL
LIN {X 0,Y 305.393,Z 1122.248,A -85,B 0,C 180,E1 5723.652,E2 5723.652} C_VEL
LIN {X 0,Y 294.972,Z 1135.07,A -85,B 0,C 180,E1 5720.307,E2 5720.307} C_VEL
LIN {X 0,Y 282.661,Z 1149.986,A -85,B 0,C 180,E1 5715.54,E2 5715.54} C_VEL
LIN {X 0,Y 273.394,Z 1161.128,A -85,B 0,C 180,E1 5711.113,E2 5711.113} C_VEL
LIN {X 0,Y 266.305,Z 1169.948,A -85,B 0,C 180,E1 5706.894,E2 5706.894} C_VEL
LIN {X 0,Y 260.17,Z 1177.992,A -85,B 0,C 180,E1 5702.273,E2 5702.273} C_VEL
LIN {X 0,Y 254.479,Z 1186.349,A -85,B 0,C 180,E1 5696.36,E2 5696.36} C_VEL
LIN {X 0,Y 250.815,Z 1192.611,A -85,B 0,C 180,E1 5690.471,E2 5690.471} C_VEL
LIN {X 0,Y 249.044,Z 1196.687,A -85,B 0,C 180,E1 5685.51,E2 5685.51} C_VEL
LIN {X 0,Y 248.223,Z 1199.509,A -85,B 0,C 180,E1 5680.914,E2 5680.914} C_VEL
LIN {X 0,Y 247.96,Z 1201.377,A -85,B 0,C 180,E1 5676.484,E2 5676.484} C_VEL
LIN {X 0,Y 247.915,Z 1202.404,A -85,B 0,C 180,E1 5672.081,E2 5672.081} C_VEL
LIN {X 0,Y 247.914,Z 1202.599,A -85,B 0,C 180,E1 5667.689,E2 5667.689} C_VEL
LIN {X 0,Y 247.969,Z 1201.901,A -85,B 0,C 180,E1 5663.053,E2 5663.053} C_VEL
LIN {X 0,Y 248.358,Z 1200.129,A -85,B 0,C 180,E1 5658.048,E2 5658.048} C_VEL
LIN {X 0,Y 249.528,Z 1197.298,A -85,B 0,C 180,E1 5652.992,E2 5652.992} C_VEL
LIN {X 0,Y 251.673,Z 1193.52,A -85,B 0,C 180,E1 5648.072,E2 5648.072} C_VEL
LIN {X 0,Y 255.049,Z 1188.708,A -85,B 0,C 180,E1 5643.204,E2 5643.204} C_VEL
LIN {X 0,Y 259.747,Z 1182.835,A -85,B 0,C 180,E1 5638.432,E2 5638.432} C_VEL
LIN {X 0,Y 266.495,Z 1175.161,A -85,B 0,C 180,E1 5633.377,E2 5633.377} C_VEL
LIN {X 0,Y 276.955,Z 1163.903,A -85,B 0,C 180,E1 5627.538,E2 5627.538} C_VEL
LIN {X 0,Y 286.85,Z 1153.456,A -85,B 0,C 180,E1 5623.239,E2 5623.239} C_VEL
LIN {X 0,Y 297.378,Z 1142.332,A -85,B 0,C 180,E1 5619.456,E2 5619.456} C_VEL
LIN {X 0,Y 310.072,Z 1128.733,A -85,B 0,C 180,E1 5615.649,E2 5615.649} C_VEL
LIN {X 0,Y 325.023,Z 1111.937,A -85,B 0,C 180,E1 5611.891,E2 5611.891} C_VEL
LIN {X 0,Y 337.055,Z 1097.752,A -85,B 0,C 180,E1 5609.292,E2 5609.292} C_VEL
LIN {X 0,Y 349.005,Z 1082.937,A -85,B 0,C 180,E1 5607.003,E2 5607.003} C_VEL
LIN {X 0,Y 361.58,Z 1066.42,A -85,B 0,C 180,E1 5604.856,E2 5604.856} C_VEL
LIN {X 0,Y 376.755,Z 1044.894,A -85,B 0,C 180,E1 5602.549,E2 5602.549} C_VEL
LIN {X 0,Y 389.391,Z 1025.148,A -85,B 0,C 180,E1 5600.826,E2 5600.826} C_VEL
LIN {X 0,Y 399.906,Z 1007.319,A -85,B 0,C 180,E1 5599.509,E2 5599.509} C_VEL
LIN {X 0,Y 410.206,Z 988.257,A -85,B 0,C 180,E1 5598.306,E2 5598.306} C_VEL
LIN {X 0,Y 421.236,Z 965.733,A -85,B 0,C 180,E1 5597.118,E2 5597.118} C_VEL
LIN {X 0,Y 431.78,Z 940.953,A -85,B 0,C 180,E1 5596.053,E2 5596.053} C_VEL
LIN {X 0,Y 439.553,Z 920.059,A -85,B 0,C 180,E1 5595.316,E2 5595.316} C_VEL
LIN {X 0,Y 446.304,Z 899.246,A -85,B 0,C 180,E1 5594.702,E2 5594.702} C_VEL
LIN {X 0,Y 452.265,Z 877.766,A -85,B 0,C 180,E1 5594.184,E2 5594.184} C_VEL
LIN {X 0,Y 458.229,Z 851.652,A -85,B 0,C 180,E1 5593.685,E2 5593.685} C_VEL
LIN {X 0,Y 462.719,Z 823.788,A -85,B 0,C 180,E1 5593.242,E2 5593.242} C_VEL
LIN {X 0,Y 473.756,Z 721.234,A -85,B 0,C 180,E1 5591.778,E2 5591.778} C_VEL
LIN {X 0,Y 484.514,Z 620.622,A -85,B 0,C 180,E1 5590.343,E2 5590.343} C_VEL
LIN {X 0,Y 482.592,Z 616.667,A -85,B 0,C 180,E1 5587.74,E2 5587.74} C_VEL
LIN {X 0,Y 481.337,Z 612.655,A -85,B 0,C 180,E1 5582.739,E2 5582.739} C_VEL
LIN {X 0,Y 482.932,Z 617.331,A -85,B 0,C 180,E1 5577.508,E2 5577.508} C_VEL
LIN {X 0,Y 484.477,Z 620.771,A -85,B 0,C 180,E1 5575.469,E2 5575.469} C_VEL
LIN {X 0,Y 462.988,Z 820.827,A -85,B 0,C 180,E1 5572.639,E2 5572.639} C_VEL
LIN {X 0,Y 459,Z 846.249,A -85,B 0,C 180,E1 5572.238,E2 5572.238} C_VEL
LIN {X 0,Y 452.871,Z 874.079,A -85,B 0,C 180,E1 5571.699,E2 5571.699} C_VEL
LIN {X 0,Y 446.967,Z 895.66,A -85,B 0,C 180,E1 5571.166,E2 5571.166} C_VEL
LIN {X 0,Y 440.41,Z 916.113,A -85,B 0,C 180,E1 5570.556,E2 5570.556} C_VEL
LIN {X 0,Y 433.212,Z 935.74,A -85,B 0,C 180,E1 5569.857,E2 5569.857} C_VEL
LIN {X 0,Y 424.313,Z 957.201,A -85,B 0,C 180,E1 5568.947,E2 5568.947} C_VEL
LIN {X 0,Y 412.035,Z 983.031,A -85,B 0,C 180,E1 5567.614,E2 5567.614} C_VEL
LIN {X 0,Y 401.272,Z 1003.073,A -85,B 0,C 180,E1 5566.355,E2 5566.355} C_VEL
LIN {X 0,Y 391.144,Z 1020.357,A -85,B 0,C 180,E1 5565.075,E2 5565.075} C_VEL
LIN {X 0,Y 380.382,Z 1037.288,A -85,B 0,C 180,E1 5563.623,E2 5563.623} C_VEL
LIN {X 0,Y 367.995,Z 1055.369,A -85,B 0,C 180,E1 5561.792,E2 5561.792} C_VEL
LIN {X 0,Y 352.02,Z 1076.735,A -85,B 0,C 180,E1 5559.144,E2 5559.144} C_VEL
LIN {X 0,Y 339.221,Z 1092.581,A -85,B 0,C 180,E1 5556.735,E2 5556.735} C_VEL
LIN {X 0,Y 327.492,Z 1106.351,A -85,B 0,C 180,E1 5554.245,E2 5554.245} C_VEL
LIN {X 0,Y 315.559,Z 1119.738,A -85,B 0,C 180,E1 5551.364,E2 5551.364} C_VEL
LIN {X 0,Y 301.512,Z 1134.906,A -85,B 0,C 180,E1 5547.384,E2 5547.384} C_VEL
LIN {X 0,Y 289.444,Z 1147.38,A -85,B 0,C 180,E1 5543.266,E2 5543.266} C_VEL
LIN {X 0,Y 279.76,Z 1157.347,A -85,B 0,C 180,E1 5539.26,E2 5539.26} C_VEL
LIN {X 0,Y 271.2,Z 1166.231,A -85,B 0,C 180,E1 5534.936,E2 5534.936} C_VEL
LIN {X 0,Y 262.49,Z 1175.713,A -85,B 0,C 180,E1 5529.221,E2 5529.221} C_VEL
LIN {X 0,Y 256.025,Z 1183.145,A -85,B 0,C 180,E1 5523.304,E2 5523.304} C_VEL
LIN {X 0,Y 252.335,Z 1188.005,A -85,B 0,C 180,E1 5518.391,E2 5518.391} C_VEL
LIN {X 0,Y 249.994,Z 1191.707,A -85,B 0,C 180,E1 5513.575,E2 5513.575} C_VEL
LIN {X 0,Y 248.659,Z 1194.439,A -85,B 0,C 180,E1 5508.764,E2 5508.764} C_VEL
LIN {X 0,Y 248.099,Z 1196.159,A -85,B 0,C 180,E1 5504.23,E2 5504.23} C_VEL
LIN {X 0,Y 247.939,Z 1197.026,A -85,B 0,C 180,E1 5499.985,E2 5499.985} C_VEL
LIN {X 0,Y 247.911,Z 1197.168,A -85,B 0,C 180,E1 5495.786,E2 5495.786} C_VEL
LIN {X 0,Y 247.944,Z 1196.46,A -85,B 0,C 180,E1 5491.154,E2 5491.154} C_VEL
LIN {X 0,Y 248.163,Z 1194.867,A -85,B 0,C 180,E1 5486.534,E2 5486.534} C_VEL
LIN {X 0,Y 248.905,Z 1192.227,A -85,B 0,C 180,E1 5481.684,E2 5481.684} C_VEL
LIN {X 0,Y 250.457,Z 1188.594,A -85,B 0,C 180,E1 5476.846,E2 5476.846} C_VEL
LIN {X 0,Y 253.073,Z 1183.944,A -85,B 0,C 180,E1 5472.05,E2 5472.05} C_VEL
LIN {X 0,Y 256.878,Z 1178.203,A -85,B 0,C 180,E1 5467.297,E2 5467.297} C_VEL
LIN {X 0,Y 262.153,Z 1171.119,A -85,B 0,C 180,E1 5462.515,E2 5462.515} C_VEL
LIN {X 0,Y 270.237,Z 1161.15,A -85,B 0,C 180,E1 5457.05,E2 5457.05} C_VEL
LIN {X 0,Y 279.816,Z 1149.569,A -85,B 0,C 180,E1 5452.075,E2 5452.075} C_VEL
LIN {X 0,Y 288.713,Z 1139.015,A -85,B 0,C 180,E1 5448.322,E2 5448.322} C_VEL
LIN {X 0,Y 298.133,Z 1127.773,A -85,B 0,C 180,E1 5444.955,E2 5444.955} C_VEL
LIN {X 0,Y 309.553,Z 1113.865,A -85,B 0,C 180,E1 5441.463,E2 5441.463} C_VEL
LIN {X 0,Y 323.165,Z 1096.481,A -85,B 0,C 180,E1 5437.909,E2 5437.909} C_VEL
LIN {X 0,Y 334.548,Z 1081.126,A -85,B 0,C 180,E1 5435.32,E2 5435.32} C_VEL
LIN {X 0,Y 345.508,Z 1065.535,A -85,B 0,C 180,E1 5433.091,E2 5433.091} C_VEL
LIN {X 0,Y 356.555,Z 1048.847,A -85,B 0,C 180,E1 5431.064,E2 5431.064} C_VEL
LIN {X 0,Y 369.893,Z 1027.133,A -85,B 0,C 180,E1 5428.857,E2 5428.857} C_VEL
LIN {X 0,Y 381.368,Z 1006.394,A -85,B 0,C 180,E1 5427.129,E2 5427.129} C_VEL
LIN {X 0,Y 390.935,Z 987.552,A -85,B 0,C 180,E1 5425.802,E2 5425.802} C_VEL
LIN {X 0,Y 399.447,Z 969.123,A -85,B 0,C 180,E1 5424.68,E2 5424.68} C_VEL
LIN {X 0,Y 407.627,Z 949.61,A -85,B 0,C 180,E1 5423.67,E2 5423.67} C_VEL
LIN {X 0,Y 416.938,Z 924.632,A -85,B 0,C 180,E1 5422.588,E2 5422.588} C_VEL
LIN {X 0,Y 424.826,Z 899.181,A -85,B 0,C 180,E1 5421.706,E2 5421.706} C_VEL
LIN {X 0,Y 430.53,Z 877.54,A -85,B 0,C 180,E1 5421.095,E2 5421.095} C_VEL
LIN {X 0,Y 435.289,Z 855.892,A -85,B 0,C 180,E1 5420.602,E2 5420.602} C_VEL
LIN {X 0,Y 439.954,Z 828.827,A -85,B 0,C 180,E1 5420.107,E2 5420.107} C_VEL
LIN {X 0,Y 443.655,Z 794.3,A -85,B 0,C 180,E1 5419.576,E2 5419.576} C_VEL
LIN {X 0,Y 444.095,Z 786.762,A -85,B 0,C 180,E1 5419.342,E2 5419.342} C_VEL
LIN {X 0,Y 444.295,Z 767.189,A -85,B 0,C 180,E1 5418.276,E2 5418.276} C_VEL
LIN {X 0,Y 444.725,Z 760.708,A -85,B 0,C 180,E1 5418.085,E2 5418.085} C_VEL
LIN {X 0,Y 459.601,Z 609.656,A -85,B 0,C 180,E1 5415.881,E2 5415.881} C_VEL
LIN {X 0,Y 456.19,Z 603.085,A -85,B 0,C 180,E1 5413.241,E2 5413.241} C_VEL
LIN {X 0,Y 454.308,Z 599.513,A -85,B 0,C 180,E1 5411.425,E2 5411.425} C_VEL
LIN {X 0,Y 452.592,Z 596.108,A -85,B 0,C 180,E1 5409.281,E2 5409.281} C_VEL
LIN {X 0,Y 450.822,Z 591.925,A -85,B 0,C 180,E1 5405.345,E2 5405.345} C_VEL
LIN {X 0,Y 450.86,Z 591.937,A -85,B 0,C 180,E1 5400.635,E2 5400.635} C_VEL
LIN {X 0,Y 452.581,Z 596.132,A -85,B 0,C 180,E1 5396.834,E2 5396.834} C_VEL
LIN {X 0,Y 453.772,Z 598.641,A -85,B 0,C 180,E1 5395.26,E2 5395.26} C_VEL
LIN {X 0,Y 455.475,Z 601.742,A -85,B 0,C 180,E1 5393.508,E2 5393.508} C_VEL
LIN {X 0,Y 457.735,Z 606.147,A -85,B 0,C 180,E1 5391.584,E2 5391.584} C_VEL
LIN {X 0,Y 459.637,Z 610.05,A -85,B 0,C 180,E1 5390.176,E2 5390.176} C_VEL
LIN {X 0,Y 438.851,Z 820.283,A -85,B 0,C 180,E1 5387.105,E2 5387.105} C_VEL
LIN {X 0,Y 435.728,Z 842.515,A -85,B 0,C 180,E1 5386.738,E2 5386.738} C_VEL
LIN {X 0,Y 431.064,Z 866.926,A -85,B 0,C 180,E1 5386.279,E2 5386.279} C_VEL
LIN {X 0,Y 424.254,Z 894.401,A -85,B 0,C 180,E1 5385.614,E2 5385.614} C_VEL
LIN {X 0,Y 417.566,Z 916.632,A -85,B 0,C 180,E1 5384.929,E2 5384.929} C_VEL
LIN {X 0,Y 410.424,Z 937.233,A -85,B 0,C 180,E1 5384.165,E2 5384.165} C_VEL
LIN {X 0,Y 402.448,Z 957.599,A -85,B 0,C 180,E1 5383.266,E2 5383.266} C_VEL
LIN {X 0,Y 391.694,Z 982.061,A -85,B 0,C 180,E1 5381.968,E2 5381.968} C_VEL
LIN {X 0,Y 379.886,Z 1005.421,A -85,B 0,C 180,E1 5380.438,E2 5380.438} C_VEL
LIN {X 0,Y 369.956,Z 1023.406,A -85,B 0,C 180,E1 5379.033,E2 5379.033} C_VEL
LIN {X 0,Y 359.85,Z 1040.308,A -85,B 0,C 180,E1 5377.502,E2 5377.502} C_VEL
LIN {X 0,Y 348.154,Z 1058.503,A -85,B 0,C 180,E1 5375.562,E2 5375.562} C_VEL
LIN {X 0,Y 332.987,Z 1080.253,A -85,B 0,C 180,E1 5372.725,E2 5372.725} C_VEL
LIN {X 0,Y 321.313,Z 1095.828,A -85,B 0,C 180,E1 5370.252,E2 5370.252} C_VEL
LIN {X 0,Y 310.254,Z 1109.893,A -85,B 0,C 180,E1 5367.605,E2 5367.605} C_VEL
LIN {X 0,Y 298.692,Z 1124.037,A -85,B 0,C 180,E1 5364.435,E2 5364.435} C_VEL
LIN {X 0,Y 284.868,Z 1140.35,A -85,B 0,C 180,E1 5359.923,E2 5359.923} C_VEL
LIN {X 0,Y 274.565,Z 1152.212,A -85,B 0,C 180,E1 5355.842,E2 5355.842} C_VEL
LIN {X 0,Y 265.967,Z 1162.175,A -85,B 0,C 180,E1 5351.715,E2 5351.715} C_VEL
LIN {X 0,Y 258.237,Z 1171.416,A -85,B 0,C 180,E1 5347.095,E2 5347.095} C_VEL
LIN {X 0,Y 250.296,Z 1181.518,A -85,B 0,C 180,E1 5340.753,E2 5340.753} C_VEL
LIN {X 0,Y 245.586,Z 1188.25,A -85,B 0,C 180,E1 5335.31,E2 5335.31} C_VEL
LIN {X 0,Y 242.783,Z 1193.025,A -85,B 0,C 180,E1 5330.492,E2 5330.492} C_VEL
LIN {X 0,Y 241.064,Z 1196.804,A -85,B 0,C 180,E1 5325.642,E2 5325.642} C_VEL
LIN {X 0,Y 240.205,Z 1199.627,A -85,B 0,C 180,E1 5320.768,E2 5320.768} C_VEL
LIN {X 0,Y 239.959,Z 1201.335,A -85,B 0,C 180,E1 5316.461,E2 5316.461} C_VEL
LIN {X 0,Y 239.915,Z 1202.309,A -85,B 0,C 180,E1 5312.151,E2 5312.151} C_VEL
LIN {X 0,Y 239.914,Z 1202.519,A -85,B 0,C 180,E1 5307.612,E2 5307.612} C_VEL
LIN {X 0,Y 239.987,Z 1201.766,A -85,B 0,C 180,E1 5302.575,E2 5302.575} C_VEL
LIN {X 0,Y 240.431,Z 1200.015,A -85,B 0,C 180,E1 5297.512,E2 5297.512} C_VEL
LIN {X 0,Y 241.7,Z 1197.264,A -85,B 0,C 180,E1 5292.424,E2 5292.424} C_VEL
LIN {X 0,Y 244.163,Z 1193.318,A -85,B 0,C 180,E1 5287.134,E2 5287.134} C_VEL
LIN {X 0,Y 247.9,Z 1188.397,A -85,B 0,C 180,E1 5282.047,E2 5282.047} C_VEL
LIN {X 0,Y 253.219,Z 1182.248,A -85,B 0,C 180,E1 5276.982,E2 5276.982} C_VEL
LIN {X 0,Y 261.957,Z 1173.047,A -85,B 0,C 180,E1 5270.966,E2 5270.966} C_VEL
LIN {X 0,Y 272.144,Z 1162.615,A -85,B 0,C 180,E1 5265.729,E2 5265.729} C_VEL
LIN {X 0,Y 282.168,Z 1152.537,A -85,B 0,C 180,E1 5261.611,E2 5261.611} C_VEL
LIN {X 0,Y 293.077,Z 1141.494,A -85,B 0,C 180,E1 5257.887,E2 5257.887} C_VEL
LIN {X 0,Y 307.627,Z 1126.457,A -85,B 0,C 180,E1 5253.767,E2 5253.767} C_VEL
LIN {X 0,Y 321.472,Z 1111.277,A -85,B 0,C 180,E1 5250.464,E2 5250.464} C_VEL
LIN {X 0,Y 333.792,Z 1097.151,A -85,B 0,C 180,E1 5247.913,E2 5247.913} C_VEL
LIN {X 0,Y 346.076,Z 1082.29,A -85,B 0,C 180,E1 5245.656,E2 5245.656} C_VEL
LIN {X 0,Y 359.634,Z 1064.852,A -85,B 0,C 180,E1 5243.441,E2 5243.441} C_VEL
LIN {X 0,Y 375.282,Z 1042.879,A -85,B 0,C 180,E1 5241.172,E2 5241.172} C_VEL
LIN {X 0,Y 387.387,Z 1024.261,A -85,B 0,C 180,E1 5239.596,E2 5239.596} C_VEL
LIN {X 0,Y 397.696,Z 1007.073,A -85,B 0,C 180,E1 5238.362,E2 5238.362} C_VEL
LIN {X 0,Y 408.171,Z 987.997,A -85,B 0,C 180,E1 5237.186,E2 5237.186} C_VEL
LIN {X 0,Y 419.694,Z 964.805,A -85,B 0,C 180,E1 5235.996,E2 5235.996} C_VEL
LIN {X 0,Y 430.077,Z 940.629,A -85,B 0,C 180,E1 5234.989,E2 5234.989} C_VEL
LIN {X 0,Y 438.15,Z 919.15,A -85,B 0,C 180,E1 5234.254,E2 5234.254} C_VEL
LIN {X 0,Y 444.897,Z 898.529,A -85,B 0,C 180,E1 5233.667,E2 5233.667} C_VEL
LIN {X 0,Y 451.169,Z 876.062,A -85,B 0,C 180,E1 5233.146,E2 5233.146} C_VEL
LIN {X 0,Y 457.532,Z 847.491,A -85,B 0,C 180,E1 5232.628,E2 5232.628} C_VEL
LIN {X 0,Y 461.493,Z 822.471,A -85,B 0,C 180,E1 5232.241,E2 5232.241} C_VEL
LIN {X 0,Y 482.786,Z 627.441,A -85,B 0,C 180,E1 5229.51,E2 5229.51} C_VEL
LIN {X 0,Y 481.545,Z 624.556,A -85,B 0,C 180,E1 5227.637,E2 5227.637} C_VEL
LIN {X 0,Y 480.353,Z 620.652,A -85,B 0,C 180,E1 5222.744,E2 5222.744} C_VEL
LIN {X 0,Y 481.865,Z 625.224,A -85,B 0,C 180,E1 5217.621,E2 5217.621} C_VEL
LIN {X 0,Y 482.75,Z 627.444,A -85,B 0,C 180,E1 5216.322,E2 5216.322} C_VEL
LIN {X 0,Y 461.595,Z 820.94,A -85,B 0,C 180,E1 5213.618,E2 5213.618} C_VEL
LIN {X 0,Y 457.528,Z 846.483,A -85,B 0,C 180,E1 5213.223,E2 5213.223} C_VEL
LIN {X 0,Y 451.318,Z 874.268,A -85,B 0,C 180,E1 5212.698,E2 5212.698} C_VEL
LIN {X 0,Y 445.334,Z 895.841,A -85,B 0,C 180,E1 5212.178,E2 5212.178} C_VEL
LIN {X 0,Y 438.667,Z 916.345,A -85,B 0,C 180,E1 5211.582,E2 5211.582} C_VEL
LIN {X 0,Y 431.37,Z 935.952,A -85,B 0,C 180,E1 5210.901,E2 5210.901} C_VEL
LIN {X 0,Y 422.342,Z 957.397,A -85,B 0,C 180,E1 5210.014,E2 5210.014} C_VEL
LIN {X 0,Y 409.875,Z 983.197,A -85,B 0,C 180,E1 5208.711,E2 5208.711} C_VEL
LIN {X 0,Y 398.935,Z 1003.226,A -85,B 0,C 180,E1 5207.478,E2 5207.478} C_VEL
LIN {X 0,Y 388.622,Z 1020.502,A -85,B 0,C 180,E1 5206.227,E2 5206.227} C_VEL
LIN {X 0,Y 377.239,Z 1038.048,A -85,B 0,C 180,E1 5204.746,E2 5204.746} C_VEL
LIN {X 0,Y 363.305,Z 1057.899,A -85,B 0,C 180,E1 5202.744,E2 5202.744} C_VEL
LIN {X 0,Y 347.892,Z 1077.799,A -85,B 0,C 180,E1 5200.263,E2 5200.263} C_VEL
LIN {X 0,Y 335.404,Z 1092.85,A -85,B 0,C 180,E1 5197.989,E2 5197.989} C_VEL
LIN {X 0,Y 323.124,Z 1106.851,A -85,B 0,C 180,E1 5195.47,E2 5195.47} C_VEL
LIN {X 0,Y 310.172,Z 1120.915,A -85,B 0,C 180,E1 5192.434,E2 5192.434} C_VEL
LIN {X 0,Y 294.513,Z 1137.048,A -85,B 0,C 180,E1 5188.075,E2 5188.075} C_VEL
LIN {X 0,Y 283.242,Z 1148.262,A -85,B 0,C 180,E1 5184.283,E2 5184.283} C_VEL
LIN {X 0,Y 273.68,Z 1157.673,A -85,B 0,C 180,E1 5180.431,E2 5180.431} C_VEL
LIN {X 0,Y 264.476,Z 1166.768,A -85,B 0,C 180,E1 5175.914,E2 5175.914} C_VEL
LIN {X 0,Y 254.897,Z 1176.572,A -85,B 0,C 180,E1 5169.745,E2 5169.745} C_VEL
LIN {X 0,Y 248.746,Z 1183.262,A -85,B 0,C 180,E1 5164.245,E2 5164.245} C_VEL
LIN {X 0,Y 244.712,Z 1188.199,A -85,B 0,C 180,E1 5159.092,E2 5159.092} C_VEL
LIN {X 0,Y 242.187,Z 1191.877,A -85,B 0,C 180,E1 5154.124,E2 5154.124} C_VEL
LIN {X 0,Y 240.732,Z 1194.585,A -85,B 0,C 180,E1 5149.154,E2 5149.154} C_VEL
LIN {X 0,Y 240.117,Z 1196.282,A -85,B 0,C 180,E1 5144.467,E2 5144.467} C_VEL
LIN {X 0,Y 239.941,Z 1197.126,A -85,B 0,C 180,E1 5140.079,E2 5140.079} C_VEL
LIN {X 0,Y 239.911,Z 1197.244,A -85,B 0,C 180,E1 5135.74,E2 5135.74} C_VEL
LIN {X 0,Y 239.944,Z 1196.581,A -85,B 0,C 180,E1 5131.193,E2 5131.193} C_VEL
LIN {X 0,Y 240.195,Z 1194.898,A -85,B 0,C 180,E1 5126.18,E2 5126.18} C_VEL
LIN {X 0,Y 241.019,Z 1192.237,A -85,B 0,C 180,E1 5121.17,E2 5121.17} C_VEL
LIN {X 0,Y 242.722,Z 1188.582,A -85,B 0,C 180,E1 5116.176,E2 5116.176} C_VEL
LIN {X 0,Y 245.544,Z 1183.908,A -85,B 0,C 180,E1 5111.234,E2 5111.234} C_VEL
LIN {X 0,Y 249.598,Z 1178.188,A -85,B 0,C 180,E1 5106.384,E2 5106.384} C_VEL
LIN {X 0,Y 255.25,Z 1171.035,A -85,B 0,C 180,E1 5101.451,E2 5101.451} C_VEL
LIN {X 0,Y 264.175,Z 1160.565,A -85,B 0,C 180,E1 5095.67,E2 5095.67} C_VEL
LIN {X 0,Y 273.861,Z 1149.403,A -85,B 0,C 180,E1 5090.829,E2 5090.829} C_VEL
LIN {X 0,Y 283.169,Z 1138.819,A -85,B 0,C 180,E1 5087.039,E2 5087.039} C_VEL
LIN {X 0,Y 293.519,Z 1126.923,A -85,B 0,C 180,E1 5083.481,E2 5083.481} C_VEL
LIN {X 0,Y 306.604,Z 1111.516,A -85,B 0,C 180,E1 5079.679,E2 5079.679} C_VEL
LIN {X 0,Y 319.515,Z 1095.315,A -85,B 0,C 180,E1 5076.462,E2 5076.462} C_VEL
LIN {X 0,Y 330.776,Z 1080.514,A -85,B 0,C 180,E1 5074.003,E2 5074.003} C_VEL
LIN {X 0,Y 342.217,Z 1064.604,A -85,B 0,C 180,E1 5071.762,E2 5071.762} C_VEL
LIN {X 0,Y 355.041,Z 1045.597,A -85,B 0,C 180,E1 5069.515,E2 5069.515} C_VEL
LIN {X 0,Y 368.328,Z 1023.911,A -85,B 0,C 180,E1 5067.415,E2 5067.415} C_VEL
LIN {X 0,Y 378.971,Z 1004.917,A -85,B 0,C 180,E1 5065.881,E2 5065.881} C_VEL
LIN {X 0,Y 388.311,Z 986.781,A -85,B 0,C 180,E1 5064.638,E2 5064.638} C_VEL
LIN {X 0,Y 397.385,Z 967.373,A -85,B 0,C 180,E1 5063.489,E2 5063.489} C_VEL
LIN {X 0,Y 407.444,Z 943.457,A -85,B 0,C 180,E1 5062.306,E2 5062.306} C_VEL
LIN {X 0,Y 416.406,Z 918.321,A -85,B 0,C 180,E1 5061.303,E2 5061.303} C_VEL
LIN {X 0,Y 423.002,Z 896.95,A -85,B 0,C 180,E1 5060.601,E2 5060.601} C_VEL
LIN {X 0,Y 428.639,Z 875.558,A -85,B 0,C 180,E1 5060.022,E2 5060.022} C_VEL
LIN {X 0,Y 434.054,Z 850.656,A -85,B 0,C 180,E1 5059.482,E2 5059.482} C_VEL
LIN {X 0,Y 438.481,Z 822.314,A -85,B 0,C 180,E1 5059,E2 5059} C_VEL
LIN {X 0,Y 444.725,Z 760.708,A -85,B 0,C 180,E1 5058.085,E2 5058.085} C_VEL
LIN {X 0,Y 445.202,Z 753.176,A -85,B 0,C 180,E1 5057.848,E2 5057.848} C_VEL
LIN {X 0,Y 445.606,Z 733.615,A -85,B 0,C 180,E1 5056.783,E2 5056.783} C_VEL
LIN {X 0,Y 446.074,Z 727.136,A -85,B 0,C 180,E1 5056.594,E2 5056.594} C_VEL
LIN {X 0,Y 457.324,Z 615.431,A -85,B 0,C 180,E1 5054.984,E2 5054.984} C_VEL
LIN {X 0,Y 454.377,Z 609.742,A -85,B 0,C 180,E1 5052.519,E2 5052.519} C_VEL
LIN {X 0,Y 452.977,Z 607.03,A -85,B 0,C 180,E1 5051.072,E2 5051.072} C_VEL
LIN {X 0,Y 451.528,Z 603.993,A -85,B 0,C 180,E1 5049.175,E2 5049.175} C_VEL
LIN {X 0,Y 449.807,Z 599.85,A -85,B 0,C 180,E1 5045.213,E2 5045.213} C_VEL
LIN {X 0,Y 449.873,Z 599.951,A -85,B 0,C 180,E1 5040.637,E2 5040.637} C_VEL
LIN {X 0,Y 451.599,Z 604.12,A -85,B 0,C 180,E1 5036.827,E2 5036.827} C_VEL
LIN {X 0,Y 454.149,Z 609.282,A -85,B 0,C 180,E1 5033.807,E2 5033.807} C_VEL
LIN {X 0,Y 456.487,Z 613.981,A -85,B 0,C 180,E1 5031.751,E2 5031.751} C_VEL
LIN {X 0,Y 457.359,Z 615.747,A -85,B 0,C 180,E1 5031.076,E2 5031.076} C_VEL
LIN {X 0,Y 436.583,Z 821.608,A -85,B 0,C 180,E1 5028.097,E2 5028.097} C_VEL
LIN {X 0,Y 433.248,Z 844.449,A -85,B 0,C 180,E1 5027.724,E2 5027.724} C_VEL
LIN {X 0,Y 427.561,Z 872.616,A -85,B 0,C 180,E1 5027.189,E2 5027.189} C_VEL
LIN {X 0,Y 421.263,Z 896.676,A -85,B 0,C 180,E1 5026.593,E2 5026.593} C_VEL
LIN {X 0,Y 414.85,Z 917.497,A -85,B 0,C 180,E1 5025.957,E2 5025.957} C_VEL
LIN {X 0,Y 407.74,Z 937.619,A -85,B 0,C 180,E1 5025.224,E2 5025.224} C_VEL
LIN {X 0,Y 399.375,Z 958.578,A -85,B 0,C 180,E1 5024.312,E2 5024.312} C_VEL
LIN {X 0,Y 387.949,Z 983.824,A -85,B 0,C 180,E1 5022.979,E2 5022.979} C_VEL
LIN {X 0,Y 376.98,Z 1005.13,A -85,B 0,C 180,E1 5021.601,E2 5021.601} C_VEL
LIN {X 0,Y 367.15,Z 1022.626,A -85,B 0,C 180,E1 5020.263,E2 5020.263} C_VEL
LIN {X 0,Y 356.729,Z 1039.738,A -85,B 0,C 180,E1 5018.745,E2 5018.745} C_VEL
LIN {X 0,Y 345.006,Z 1057.621,A -85,B 0,C 180,E1 5016.872,E2 5016.872} C_VEL
LIN {X 0,Y 330.466,Z 1078.162,A -85,B 0,C 180,E1 5014.269,E2 5014.269} C_VEL
LIN {X 0,Y 317.212,Z 1095.407,A -85,B 0,C 180,E1 5011.575,E2 5011.575} C_VEL
LIN {X 0,Y 305.812,Z 1109.504,A -85,B 0,C 180,E1 5008.941,E2 5008.941} C_VEL
LIN {X 0,Y 294.459,Z 1122.961,A -85,B 0,C 180,E1 5005.95,E2 5005.95} C_VEL
LIN {X 0,Y 281.124,Z 1138.278,A -85,B 0,C 180,E1 5001.817,E2 5001.817} C_VEL
LIN {X 0,Y 269.236,Z 1151.401,A -85,B 0,C 180,E1 4997.336,E2 4997.336} C_VEL
LIN {X 0,Y 260.154,Z 1161.442,A -85,B 0,C 180,E1 4993.168,E2 4993.168} C_VEL
LIN {X 0,Y 252.141,Z 1170.491,A -85,B 0,C 180,E1 4988.627,E2 4988.627} C_VEL
LIN {X 0,Y 244.469,Z 1179.696,A -85,B 0,C 180,E1 4982.955,E2 4982.955} C_VEL
LIN {X 0,Y 238.469,Z 1187.548,A -85,B 0,C 180,E1 4976.657,E2 4976.657} C_VEL
LIN {X 0,Y 235.152,Z 1192.71,A -85,B 0,C 180,E1 4971.375,E2 4971.375} C_VEL
LIN {X 0,Y 233.193,Z 1196.659,A -85,B 0,C 180,E1 4966.184,E2 4966.184} C_VEL
LIN {X 0,Y 232.245,Z 1199.485,A -85,B 0,C 180,E1 4961.172,E2 4961.172} C_VEL
LIN {X 0,Y 231.964,Z 1201.224,A -85,B 0,C 180,E1 4956.684,E2 4956.684} C_VEL
LIN {X 0,Y 231.916,Z 1202.236,A -85,B 0,C 180,E1 4951.978,E2 4951.978} C_VEL
LIN {X 0,Y 231.915,Z 1202.416,A -85,B 0,C 180,E1 4947.283,E2 4947.283} C_VEL
LIN {X 0,Y 232.002,Z 1201.702,A -85,B 0,C 180,E1 4942.323,E2 4942.323} C_VEL
LIN {X 0,Y 232.497,Z 1199.965,A -85,B 0,C 180,E1 4937.079,E2 4937.079} C_VEL
LIN {X 0,Y 233.889,Z 1197.23,A -85,B 0,C 180,E1 4931.817,E2 4931.817} C_VEL
LIN {X 0,Y 236.585,Z 1193.278,A -85,B 0,C 180,E1 4926.329,E2 4926.329} C_VEL
LIN {X 0,Y 240.533,Z 1188.454,A -85,B 0,C 180,E1 4921.172,E2 4921.172} C_VEL
LIN {X 0,Y 245.957,Z 1182.571,A -85,B 0,C 180,E1 4916.157,E2 4916.157} C_VEL
LIN {X 0,Y 253.972,Z 1174.534,A -85,B 0,C 180,E1 4910.667,E2 4910.667} C_VEL
LIN {X 0,Y 265.731,Z 1163.151,A -85,B 0,C 180,E1 4904.672,E2 4904.672} C_VEL
LIN {X 0,Y 276.14,Z 1153.15,A -85,B 0,C 180,E1 4900.503,E2 4900.503} C_VEL
LIN {X 0,Y 287.42,Z 1142.198,A -85,B 0,C 180,E1 4896.753,E2 4896.753} C_VEL
LIN {X 0,Y 300.007,Z 1129.665,A -85,B 0,C 180,E1 4893.225,E2 4893.225} C_VEL
LIN {X 0,Y 316.776,Z 1112.108,A -85,B 0,C 180,E1 4889.292,E2 4889.292} C_VEL
LIN {X 0,Y 330.002,Z 1097.385,A -85,B 0,C 180,E1 4886.643,E2 4886.643} C_VEL
LIN {X 0,Y 342.587,Z 1082.556,A -85,B 0,C 180,E1 4884.413,E2 4884.413} C_VEL
LIN {X 0,Y 355.663,Z 1066.157,A -85,B 0,C 180,E1 4882.346,E2 4882.346} C_VEL
LIN {X 0,Y 371.85,Z 1044.098,A -85,B 0,C 180,E1 4880.076,E2 4880.076} C_VEL
LIN {X 0,Y 384.738,Z 1024.691,A -85,B 0,C 180,E1 4878.456,E2 4878.456} C_VEL
LIN {X 0,Y 395.697,Z 1006.748,A -85,B 0,C 180,E1 4877.197,E2 4877.197} C_VEL
LIN {X 0,Y 406.294,Z 987.743,A -85,B 0,C 180,E1 4876.055,E2 4876.055} C_VEL
LIN {X 0,Y 418.43,Z 963.626,A -85,B 0,C 180,E1 4874.855,E2 4874.855} C_VEL
LIN {X 0,Y 428.725,Z 939.803,A -85,B 0,C 180,E1 4873.9,E2 4873.9} C_VEL
LIN {X 0,Y 436.511,Z 919.357,A -85,B 0,C 180,E1 4873.221,E2 4873.221} C_VEL
LIN {X 0,Y 443.262,Z 899.051,A -85,B 0,C 180,E1 4872.657,E2 4872.657} C_VEL
LIN {X 0,Y 449.351,Z 877.658,A -85,B 0,C 180,E1 4872.17,E2 4872.17} C_VEL
LIN {X 0,Y 455.434,Z 851.666,A -85,B 0,C 180,E1 4871.7,E2 4871.7} C_VEL
LIN {X 0,Y 460.065,Z 823.79,A -85,B 0,C 180,E1 4871.273,E2 4871.273} C_VEL
LIN {X 0,Y 470.595,Z 729.538,A -85,B 0,C 180,E1 4869.962,E2 4869.962} C_VEL
LIN {X 0,Y 481.148,Z 634.117,A -85,B 0,C 180,E1 4868.635,E2 4868.635} C_VEL
LIN {X 0,Y 480.429,Z 632.361,A -85,B 0,C 180,E1 4867.414,E2 4867.414} C_VEL
LIN {X 0,Y 479.37,Z 628.647,A -85,B 0,C 180,E1 4862.75,E2 4862.75} C_VEL
LIN {X 0,Y 480.801,Z 633.115,A -85,B 0,C 180,E1 4857.735,E2 4857.735} C_VEL
LIN {X 0,Y 481.128,Z 634.137,A -85,B 0,C 180,E1 4857.181,E2 4857.181} C_VEL
LIN {X 0,Y 460.338,Z 821.054,A -85,B 0,C 180,E1 4854.603,E2 4854.603} C_VEL
LIN {X 0,Y 456.192,Z 846.731,A -85,B 0,C 180,E1 4854.213,E2 4854.213} C_VEL
LIN {X 0,Y 449.904,Z 874.478,A -85,B 0,C 180,E1 4853.703,E2 4853.703} C_VEL
LIN {X 0,Y 443.817,Z 896.126,A -85,B 0,C 180,E1 4853.195,E2 4853.195} C_VEL
LIN {X 0,Y 437.113,Z 916.461,A -85,B 0,C 180,E1 4852.619,E2 4852.619} C_VEL
LIN {X 0,Y 429.465,Z 936.69,A -85,B 0,C 180,E1 4851.934,E2 4851.934} C_VEL
LIN {X 0,Y 419.158,Z 960.683,A -85,B 0,C 180,E1 4850.953,E2 4850.953} C_VEL
LIN {X 0,Y 406.97,Z 985.03,A -85,B 0,C 180,E1 4849.726,E2 4849.726} C_VEL
LIN {X 0,Y 396.313,Z 1004.139,A -85,B 0,C 180,E1 4848.566,E2 4848.566} C_VEL
LIN {X 0,Y 385.828,Z 1021.331,A -85,B 0,C 180,E1 4847.341,E2 4847.341} C_VEL
LIN {X 0,Y 373.822,Z 1039.431,A -85,B 0,C 180,E1 4845.832,E2 4845.832} C_VEL
LIN {X 0,Y 358.398,Z 1060.727,A -85,B 0,C 180,E1 4843.677,E2 4843.677} C_VEL
LIN {X 0,Y 343.901,Z 1078.863,A -85,B 0,C 180,E1 4841.409,E2 4841.409} C_VEL
LIN {X 0,Y 331.513,Z 1093.396,A -85,B 0,C 180,E1 4839.224,E2 4839.224} C_VEL
LIN {X 0,Y 318.909,Z 1107.354,A -85,B 0,C 180,E1 4836.727,E2 4836.727} C_VEL
LIN {X 0,Y 304.224,Z 1122.807,A -85,B 0,C 180,E1 4833.374,E2 4833.374} C_VEL
LIN {X 0,Y 289.388,Z 1137.44,A -85,B 0,C 180,E1 4829.352,E2 4829.352} C_VEL
LIN {X 0,Y 277.684,Z 1148.62,A -85,B 0,C 180,E1 4825.544,E2 4825.544} C_VEL
LIN {X 0,Y 267.716,Z 1158.002,A -85,B 0,C 180,E1 4821.656,E2 4821.656} C_VEL
LIN {X 0,Y 257.657,Z 1167.478,A -85,B 0,C 180,E1 4816.848,E2 4816.848} C_VEL
LIN {X 0,Y 247.647,Z 1177.124,A -85,B 0,C 180,E1 4810.543,E2 4810.543} C_VEL
LIN {X 0,Y 241.436,Z 1183.482,A -85,B 0,C 180,E1 4805.144,E2 4805.144} C_VEL
LIN {X 0,Y 237.124,Z 1188.395,A -85,B 0,C 180,E1 4799.838,E2 4799.838} C_VEL
LIN {X 0,Y 234.386,Z 1192.068,A -85,B 0,C 180,E1 4794.679,E2 4794.679} C_VEL
LIN {X 0,Y 232.812,Z 1194.732,A -85,B 0,C 180,E1 4789.571,E2 4789.571} C_VEL
LIN {X 0,Y 232.138,Z 1196.405,A -85,B 0,C 180,E1 4784.721,E2 4784.721} C_VEL
LIN {X 0,Y 231.943,Z 1197.225,A -85,B 0,C 180,E1 4780.179,E2 4780.179} C_VEL
LIN {X 0,Y 231.913,Z 1197.343,A -85,B 0,C 180,E1 4775.938,E2 4775.938} C_VEL
LIN {X 0,Y 231.949,Z 1196.634,A -85,B 0,C 180,E1 4770.987,E2 4770.987} C_VEL
LIN {X 0,Y 232.207,Z 1195.041,A -85,B 0,C 180,E1 4766.049,E2 4766.049} C_VEL
LIN {X 0,Y 233.086,Z 1192.402,A -85,B 0,C 180,E1 4760.866,E2 4760.866} C_VEL
LIN {X 0,Y 234.904,Z 1188.77,A -85,B 0,C 180,E1 4755.706,E2 4755.706} C_VEL
LIN {X 0,Y 237.89,Z 1184.12,A -85,B 0,C 180,E1 4750.606,E2 4750.606} C_VEL
LIN {X 0,Y 242.179,Z 1178.424,A -85,B 0,C 180,E1 4745.614,E2 4745.614} C_VEL
LIN {X 0,Y 248.128,Z 1171.295,A -85,B 0,C 180,E1 4740.552,E2 4740.552} C_VEL
LIN {X 0,Y 257.101,Z 1161.323,A -85,B 0,C 180,E1 4734.859,E2 4734.859} C_VEL
LIN {X 0,Y 267.587,Z 1149.74,A -85,B 0,C 180,E1 4729.725,E2 4729.725} C_VEL
LIN {X 0,Y 277.463,Z 1138.961,A -85,B 0,C 180,E1 4725.819,E2 4725.819} C_VEL
LIN {X 0,Y 287.976,Z 1127.313,A -85,B 0,C 180,E1 4722.306,E2 4722.306} C_VEL
LIN {X 0,Y 301.478,Z 1111.958,A -85,B 0,C 180,E1 4718.489,E2 4718.489} C_VEL
LIN {X 0,Y 315.412,Z 1094.97,A -85,B 0,C 180,E1 4715.126,E2 4715.126} C_VEL
LIN {X 0,Y 326.839,Z 1080.35,A -85,B 0,C 180,E1 4712.723,E2 4712.723} C_VEL
LIN {X 0,Y 338.039,Z 1065.16,A -85,B 0,C 180,E1 4710.599,E2 4710.599} C_VEL
LIN {X 0,Y 350.027,Z 1047.824,A -85,B 0,C 180,E1 4708.55,E2 4708.55} C_VEL
LIN {X 0,Y 364.706,Z 1024.603,A -85,B 0,C 180,E1 4706.297,E2 4706.297} C_VEL
LIN {X 0,Y 375.548,Z 1005.668,A -85,B 0,C 180,E1 4704.783,E2 4704.783} C_VEL
LIN {X 0,Y 385.451,Z 986.805,A -85,B 0,C 180,E1 4703.509,E2 4703.509} C_VEL
LIN {X 0,Y 394.686,Z 967.383,A -85,B 0,C 180,E1 4702.38,E2 4702.38} C_VEL
LIN {X 0,Y 404.912,Z 943.444,A -85,B 0,C 180,E1 4701.221,E2 4701.221} C_VEL
LIN {X 0,Y 414.013,Z 918.282,A -85,B 0,C 180,E1 4700.238,E2 4700.238} C_VEL
LIN {X 0,Y 420.709,Z 896.889,A -85,B 0,C 180,E1 4699.551,E2 4699.551} C_VEL
LIN {X 0,Y 426.416,Z 875.52,A -85,B 0,C 180,E1 4698.986,E2 4698.986} C_VEL
LIN {X 0,Y 431.977,Z 850.244,A -85,B 0,C 180,E1 4698.451,E2 4698.451} C_VEL
LIN {X 0,Y 436.395,Z 822.16,A -85,B 0,C 180,E1 4697.983,E2 4697.983} C_VEL
LIN {X 0,Y 444.83,Z 739.618,A -85,B 0,C 180,E1 4696.774,E2 4696.774} C_VEL
LIN {X 0,Y 446.074,Z 727.136,A -85,B 0,C 180,E1 4696.594,E2 4696.594} C_VEL
LIN {X 0,Y 446.595,Z 719.604,A -85,B 0,C 180,E1 4696.359,E2 4696.359} C_VEL
LIN {X 0,Y 447.202,Z 700.054,A -85,B 0,C 180,E1 4695.293,E2 4695.293} C_VEL
LIN {X 0,Y 447.713,Z 693.573,A -85,B 0,C 180,E1 4695.109,E2 4695.109} C_VEL
LIN {X 0,Y 455.126,Z 621.49,A -85,B 0,C 180,E1 4694.082,E2 4694.082} C_VEL
LIN {X 0,Y 452.353,Z 615.699,A -85,B 0,C 180,E1 4691.475,E2 4691.475} C_VEL
LIN {X 0,Y 450.376,Z 611.769,A -85,B 0,C 180,E1 4688.941,E2 4688.941} C_VEL
LIN {X 0,Y 448.803,Z 607.778,A -85,B 0,C 180,E1 4685.113,E2 4685.113} C_VEL
LIN {X 0,Y 448.863,Z 607.829,A -85,B 0,C 180,E1 4680.766,E2 4680.766} C_VEL
LIN {X 0,Y 450.525,Z 611.992,A -85,B 0,C 180,E1 4676.947,E2 4676.947} C_VEL
LIN {X 0,Y 452.957,Z 617.092,A -85,B 0,C 180,E1 4673.981,E2 4673.981} C_VEL
LIN {X 0,Y 455.166,Z 621.662,A -85,B 0,C 180,E1 4671.981,E2 4671.981} C_VEL
LIN {X 0,Y 434.471,Z 822.697,A -85,B 0,C 180,E1 4669.104,E2 4669.104} C_VEL
LIN {X 0,Y 430.703,Z 847.526,A -85,B 0,C 180,E1 4668.702,E2 4668.702} C_VEL
LIN {X 0,Y 424.529,Z 876.232,A -85,B 0,C 180,E1 4668.15,E2 4668.15} C_VEL
LIN {X 0,Y 418.697,Z 897.929,A -85,B 0,C 180,E1 4667.614,E2 4667.614} C_VEL
LIN {X 0,Y 412.247,Z 918.427,A -85,B 0,C 180,E1 4666.998,E2 4666.998} C_VEL
LIN {X 0,Y 404.89,Z 938.819,A -85,B 0,C 180,E1 4666.265,E2 4666.265} C_VEL
LIN {X 0,Y 395.029,Z 962.913,A -85,B 0,C 180,E1 4665.218,E2 4665.218} C_VEL
LIN {X 0,Y 383.477,Z 987.233,A -85,B 0,C 180,E1 4663.911,E2 4663.911} C_VEL
LIN {X 0,Y 373.436,Z 1006.262,A -85,B 0,C 180,E1 4662.683,E2 4662.683} C_VEL
LIN {X 0,Y 363.093,Z 1024.224,A -85,B 0,C 180,E1 4661.317,E2 4661.317} C_VEL
LIN {X 0,Y 351.789,Z 1042.278,A -85,B 0,C 180,E1 4659.711,E2 4659.711} C_VEL
LIN {X 0,Y 336.933,Z 1064.074,A -85,B 0,C 180,E1 4657.358,E2 4657.358} C_VEL
LIN {X 0,Y 323.767,Z 1081.715,A -85,B 0,C 180,E1 4655.014,E2 4655.014} C_VEL
LIN {X 0,Y 311.872,Z 1096.716,A -85,B 0,C 180,E1 4652.634,E2 4652.634} C_VEL
LIN {X 0,Y 299.533,Z 1111.477,A -85,B 0,C 180,E1 4649.835,E2 4649.835} C_VEL
LIN {X 0,Y 284.853,Z 1128.221,A -85,B 0,C 180,E1 4645.935,E2 4645.935} C_VEL
LIN {X 0,Y 272.052,Z 1142.063,A -85,B 0,C 180,E1 4641.869,E2 4641.869} C_VEL
LIN {X 0,Y 262.071,Z 1152.692,A -85,B 0,C 180,E1 4638.073,E2 4638.073} C_VEL
LIN {X 0,Y 252.742,Z 1162.586,A -85,B 0,C 180,E1 4633.815,E2 4633.815} C_VEL
LIN {X 0,Y 242.945,Z 1173.318,A -85,B 0,C 180,E1 4628.124,E2 4628.124} C_VEL
LIN {X 0,Y 234.992,Z 1182.355,A -85,B 0,C 180,E1 4621.845,E2 4621.845} C_VEL
LIN {X 0,Y 230.263,Z 1188.423,A -85,B 0,C 180,E1 4616.551,E2 4616.551} C_VEL
LIN {X 0,Y 227.127,Z 1193.12,A -85,B 0,C 180,E1 4611.432,E2 4611.432} C_VEL
LIN {X 0,Y 225.193,Z 1196.839,A -85,B 0,C 180,E1 4606.245,E2 4606.245} C_VEL
LIN {X 0,Y 224.229,Z 1199.589,A -85,B 0,C 180,E1 4601.056,E2 4601.056} C_VEL
LIN {X 0,Y 223.956,Z 1201.251,A -85,B 0,C 180,E1 4596.409,E2 4596.409} C_VEL
LIN {X 0,Y 223.918,Z 1202.164,A -85,B 0,C 180,E1 4591.792,E2 4591.792} C_VEL
LIN {X 0,Y 223.915,Z 1202.336,A -85,B 0,C 180,E1 4587.186,E2 4587.186} C_VEL
LIN {X 0,Y 224.009,Z 1201.637,A -85,B 0,C 180,E1 4582.047,E2 4582.047} C_VEL
LIN {X 0,Y 224.573,Z 1199.916,A -85,B 0,C 180,E1 4576.614,E2 4576.614} C_VEL
LIN {X 0,Y 226.194,Z 1197.036,A -85,B 0,C 180,E1 4570.908,E2 4570.908} C_VEL
LIN {X 0,Y 229.2,Z 1193.054,A -85,B 0,C 180,E1 4565.242,E2 4565.242} C_VEL
LIN {X 0,Y 233.772,Z 1187.947,A -85,B 0,C 180,E1 4559.69,E2 4559.69} C_VEL
LIN {X 0,Y 241.001,Z 1180.775,A -85,B 0,C 180,E1 4553.611,E2 4553.611} C_VEL
LIN {X 0,Y 251.295,Z 1171.105,A -85,B 0,C 180,E1 4547.401,E2 4547.401} C_VEL
LIN {X 0,Y 261.362,Z 1161.866,A -85,B 0,C 180,E1 4542.735,E2 4542.735} C_VEL
LIN {X 0,Y 272.439,Z 1151.724,A -85,B 0,C 180,E1 4538.582,E2 4538.582} C_VEL
LIN {X 0,Y 285.366,Z 1139.668,A -85,B 0,C 180,E1 4534.575,E2 4534.575} C_VEL
LIN {X 0,Y 301.503,Z 1123.883,A -85,B 0,C 180,E1 4530.433,E2 4530.433} C_VEL
LIN {X 0,Y 314.702,Z 1110.271,A -85,B 0,C 180,E1 4527.572,E2 4527.572} C_VEL
LIN {X 0,Y 327.12,Z 1096.79,A -85,B 0,C 180,E1 4525.212,E2 4525.212} C_VEL
LIN {X 0,Y 340.05,Z 1081.905,A -85,B 0,C 180,E1 4523.022,E2 4523.022} C_VEL
LIN {X 0,Y 354.231,Z 1064.463,A -85,B 0,C 180,E1 4520.887,E2 4520.887} C_VEL
LIN {X 0,Y 370.533,Z 1042.45,A -85,B 0,C 180,E1 4518.71,E2 4518.71} C_VEL
LIN {X 0,Y 383.087,Z 1023.812,A -85,B 0,C 180,E1 4517.203,E2 4517.203} C_VEL
LIN {X 0,Y 394.191,Z 1005.874,A -85,B 0,C 180,E1 4515.986,E2 4515.986} C_VEL
LIN {X 0,Y 404.932,Z 986.841,A -85,B 0,C 180,E1 4514.881,E2 4514.881} C_VEL
LIN {X 0,Y 417.111,Z 962.859,A -85,B 0,C 180,E1 4513.729,E2 4513.729} C_VEL
LIN {X 0,Y 427.57,Z 938.894,A -85,B 0,C 180,E1 4512.801,E2 4512.801} C_VEL
LIN {X 0,Y 435.663,Z 917.759,A -85,B 0,C 180,E1 4512.126,E2 4512.126} C_VEL
LIN {X 0,Y 442.637,Z 896.785,A -85,B 0,C 180,E1 4511.572,E2 4511.572} C_VEL
LIN {X 0,Y 449.898,Z 870.945,A -85,B 0,C 180,E1 4511.026,E2 4511.026} C_VEL
LIN {X 0,Y 455.77,Z 843.408,A -85,B 0,C 180,E1 4510.572,E2 4510.572} C_VEL
LIN {X 0,Y 459.346,Z 820.757,A -85,B 0,C 180,E1 4510.238,E2 4510.238} C_VEL
LIN {X 0,Y 479.653,Z 640.756,A -85,B 0,C 180,E1 4507.788,E2 4507.788} C_VEL
LIN {X 0,Y 478.386,Z 636.64,A -85,B 0,C 180,E1 4502.755,E2 4502.755} C_VEL
LIN {X 0,Y 479.617,Z 640.82,A -85,B 0,C 180,E1 4498.045,E2 4498.045} C_VEL
LIN {X 0,Y 459.202,Z 821.279,A -85,B 0,C 180,E1 4495.592,E2 4495.592} C_VEL
LIN {X 0,Y 454.919,Z 847.397,A -85,B 0,C 180,E1 4495.203,E2 4495.203} C_VEL
LIN {X 0,Y 448.598,Z 874.8,A -85,B 0,C 180,E1 4494.712,E2 4494.712} C_VEL
LIN {X 0,Y 442.441,Z 896.411,A -85,B 0,C 180,E1 4494.218,E2 4494.218} C_VEL
LIN {X 0,Y 435.609,Z 916.85,A -85,B 0,C 180,E1 4493.655,E2 4493.655} C_VEL
LIN {X 0,Y 427.656,Z 937.56,A -85,B 0,C 180,E1 4492.971,E2 4492.971} C_VEL
LIN {X 0,Y 417.006,Z 961.899,A -85,B 0,C 180,E1 4491.996,E2 4491.996} C_VEL
LIN {X 0,Y 405.103,Z 985.203,A -85,B 0,C 180,E1 4490.847,E2 4490.847} C_VEL
LIN {X 0,Y 394.283,Z 1004.302,A -85,B 0,C 180,E1 4489.714,E2 4489.714} C_VEL
LIN {X 0,Y 383.62,Z 1021.485,A -85,B 0,C 180,E1 4488.522,E2 4488.522} C_VEL
LIN {X 0,Y 370.97,Z 1040.195,A -85,B 0,C 180,E1 4486.992,E2 4486.992} C_VEL
LIN {X 0,Y 354,Z 1062.928,A -85,B 0,C 180,E1 4484.7,E2 4484.7} C_VEL
LIN {X 0,Y 340.455,Z 1079.46,A -85,B 0,C 180,E1 4482.645,E2 4482.645} C_VEL
LIN {X 0,Y 327.78,Z 1093.943,A -85,B 0,C 180,E1 4480.488,E2 4480.488} C_VEL
LIN {X 0,Y 314.662,Z 1108.059,A -85,B 0,C 180,E1 4477.978,E2 4477.978} C_VEL
LIN {X 0,Y 299.048,Z 1123.96,A -85,B 0,C 180,E1 4474.52,E2 4474.52} C_VEL
LIN {X 0,Y 284.414,Z 1137.834,A -85,B 0,C 180,E1 4470.674,E2 4470.674} C_VEL
LIN {X 0,Y 272.848,Z 1148.458,A -85,B 0,C 180,E1 4467.053,E2 4467.053} C_VEL
LIN {X 0,Y 262.393,Z 1157.865,A -85,B 0,C 180,E1 4463.15,E2 4463.15} C_VEL
LIN {X 0,Y 252.234,Z 1166.958,A -85,B 0,C 180,E1 4458.52,E2 4458.52} C_VEL
LIN {X 0,Y 241.474,Z 1176.758,A -85,B 0,C 180,E1 4452.127,E2 4452.127} C_VEL
LIN {X 0,Y 234.342,Z 1183.551,A -85,B 0,C 180,E1 4446.251,E2 4446.251} C_VEL
LIN {X 0,Y 229.757,Z 1188.383,A -85,B 0,C 180,E1 4440.898,E2 4440.898} C_VEL
LIN {X 0,Y 226.745,Z 1192.06,A -85,B 0,C 180,E1 4435.603,E2 4435.603} C_VEL
LIN {X 0,Y 224.957,Z 1194.766,A -85,B 0,C 180,E1 4430.284,E2 4430.284} C_VEL
LIN {X 0,Y 224.186,Z 1196.461,A -85,B 0,C 180,E1 4425.255,E2 4425.255} C_VEL
LIN {X 0,Y 223.95,Z 1197.302,A -85,B 0,C 180,E1 4420.547,E2 4420.547} C_VEL
LIN {X 0,Y 223.913,Z 1197.419,A -85,B 0,C 180,E1 4415.894,E2 4415.894} C_VEL
LIN {X 0,Y 223.949,Z 1196.754,A -85,B 0,C 180,E1 4411.022,E2 4411.022} C_VEL
LIN {X 0,Y 224.246,Z 1195.071,A -85,B 0,C 180,E1 4405.652,E2 4405.652} C_VEL
LIN {X 0,Y 225.242,Z 1192.378,A -85,B 0,C 180,E1 4400.233,E2 4400.233} C_VEL
LIN {X 0,Y 227.229,Z 1188.756,A -85,B 0,C 180,E1 4394.952,E2 4394.952} C_VEL
LIN {X 0,Y 230.449,Z 1184.084,A -85,B 0,C 180,E1 4389.689,E2 4389.689} C_VEL
LIN {X 0,Y 235.055,Z 1178.363,A -85,B 0,C 180,E1 4384.555,E2 4384.555} C_VEL
LIN {X 0,Y 241.389,Z 1171.209,A -85,B 0,C 180,E1 4379.369,E2 4379.369} C_VEL
LIN {X 0,Y 251.277,Z 1160.736,A -85,B 0,C 180,E1 4373.353,E2 4373.353} C_VEL
LIN {X 0,Y 261.897,Z 1149.57,A -85,B 0,C 180,E1 4368.37,E2 4368.37} C_VEL
LIN {X 0,Y 272.003,Z 1138.981,A -85,B 0,C 180,E1 4364.508,E2 4364.508} C_VEL
LIN {X 0,Y 283.139,Z 1127.081,A -85,B 0,C 180,E1 4360.911,E2 4360.911} C_VEL
LIN {X 0,Y 297.636,Z 1111.035,A -85,B 0,C 180,E1 4356.966,E2 4356.966} C_VEL
LIN {X 0,Y 311.482,Z 1094.625,A -85,B 0,C 180,E1 4353.756,E2 4353.756} C_VEL
LIN {X 0,Y 323.238,Z 1079.961,A -85,B 0,C 180,E1 4351.377,E2 4351.377} C_VEL
LIN {X 0,Y 334.737,Z 1064.719,A -85,B 0,C 180,E1 4349.282,E2 4349.282} C_VEL
LIN {X 0,Y 348.156,Z 1045.697,A -85,B 0,C 180,E1 4347.089,E2 4347.089} C_VEL
LIN {X 0,Y 362.008,Z 1023.987,A -85,B 0,C 180,E1 4345.048,E2 4345.048} C_VEL
LIN {X 0,Y 373.063,Z 1004.977,A -85,B 0,C 180,E1 4343.562,E2 4343.562} C_VEL
LIN {X 0,Y 383.148,Z 986.025,A -85,B 0,C 180,E1 4342.313,E2 4342.313} C_VEL
LIN {X 0,Y 392.962,Z 965.621,A -85,B 0,C 180,E1 4341.164,E2 4341.164} C_VEL
LIN {X 0,Y 404.194,Z 939.011,A -85,B 0,C 180,E1 4339.943,E2 4339.943} C_VEL
LIN {X 0,Y 412.213,Z 916.908,A -85,B 0,C 180,E1 4339.115,E2 4339.115} C_VEL
LIN {X 0,Y 418.711,Z 896.309,A -85,B 0,C 180,E1 4338.475,E2 4338.475} C_VEL
LIN {X 0,Y 424.573,Z 874.522,A -85,B 0,C 180,E1 4337.917,E2 4337.917} C_VEL
LIN {X 0,Y 430.515,Z 847.319,A -85,B 0,C 180,E1 4337.367,E2 4337.367} C_VEL
LIN {X 0,Y 434.574,Z 820.926,A -85,B 0,C 180,E1 4336.941,E2 4336.941} C_VEL
LIN {X 0,Y 447.713,Z 693.573,A -85,B 0,C 180,E1 4335.109,E2 4335.109} C_VEL
LIN {X 0,Y 448.286,Z 686.04,A -85,B 0,C 180,E1 4334.88,E2 4334.88} C_VEL
LIN {X 0,Y 449.092,Z 666.503,A -85,B 0,C 180,E1 4333.817,E2 4333.817} C_VEL
LIN {X 0,Y 449.631,Z 660.025,A -85,B 0,C 180,E1 4333.631,E2 4333.631} C_VEL
LIN {X 0,Y 453.048,Z 627.497,A -85,B 0,C 180,E1 4333.175,E2 4333.175} C_VEL
LIN {X 0,Y 450.793,Z 622.843,A -85,B 0,C 180,E1 4330.867,E2 4330.867} C_VEL
LIN {X 0,Y 449.317,Z 619.654,A -85,B 0,C 180,E1 4328.833,E2 4328.833} C_VEL
LIN {X 0,Y 447.796,Z 615.705,A -85,B 0,C 180,E1 4324.996,E2 4324.996} C_VEL
LIN {X 0,Y 447.872,Z 615.879,A -85,B 0,C 180,E1 4320.768,E2 4320.768} C_VEL
LIN {X 0,Y 449.738,Z 620.577,A -85,B 0,C 180,E1 4316.622,E2 4316.622} C_VEL
LIN {X 0,Y 451.829,Z 625.035,A -85,B 0,C 180,E1 4314.094,E2 4314.094} C_VEL
LIN {X 0,Y 453.07,Z 627.723,A -85,B 0,C 180,E1 4312.893,E2 4312.893} C_VEL
LIN {X 0,Y 432.62,Z 822.774,A -85,B 0,C 180,E1 4310.136,E2 4310.136} C_VEL
LIN {X 0,Y 428.692,Z 848.184,A -85,B 0,C 180,E1 4309.731,E2 4309.731} C_VEL
LIN {X 0,Y 422.502,Z 876.405,A -85,B 0,C 180,E1 4309.2,E2 4309.2} C_VEL
LIN {X 0,Y 416.562,Z 898.169,A -85,B 0,C 180,E1 4308.675,E2 4308.675} C_VEL
LIN {X 0,Y 410.2,Z 918.121,A -85,B 0,C 180,E1 4308.09,E2 4308.09} C_VEL
LIN {X 0,Y 402.696,Z 938.656,A -85,B 0,C 180,E1 4307.372,E2 4307.372} C_VEL
LIN {X 0,Y 392.695,Z 962.745,A -85,B 0,C 180,E1 4306.352,E2 4306.352} C_VEL
LIN {X 0,Y 380.83,Z 987.328,A -85,B 0,C 180,E1 4305.06,E2 4305.06} C_VEL
LIN {X 0,Y 370.581,Z 1006.414,A -85,B 0,C 180,E1 4303.851,E2 4303.851} C_VEL
LIN {X 0,Y 360.131,Z 1024.215,A -85,B 0,C 180,E1 4302.525,E2 4302.525} C_VEL
LIN {X 0,Y 348.164,Z 1042.949,A -85,B 0,C 180,E1 4300.882,E2 4300.882} C_VEL
LIN {X 0,Y 332.223,Z 1065.656,A -85,B 0,C 180,E1 4298.433,E2 4298.433} C_VEL
LIN {X 0,Y 319.547,Z 1082.204,A -85,B 0,C 180,E1 4296.242,E2 4296.242} C_VEL
LIN {X 0,Y 307.364,Z 1097.156,A -85,B 0,C 180,E1 4293.878,E2 4293.878} C_VEL
LIN {X 0,Y 294.694,Z 1111.873,A -85,B 0,C 180,E1 4291.091,E2 4291.091} C_VEL
LIN {X 0,Y 278.937,Z 1129.18,A -85,B 0,C 180,E1 4287.014,E2 4287.014} C_VEL
LIN {X 0,Y 266.892,Z 1141.76,A -85,B 0,C 180,E1 4283.296,E2 4283.296} C_VEL
LIN {X 0,Y 255.979,Z 1152.93,A -85,B 0,C 180,E1 4279.27,E2 4279.27} C_VEL
LIN {X 0,Y 245.814,Z 1163.259,A -85,B 0,C 180,E1 4274.725,E2 4274.725} C_VEL
LIN {X 0,Y 234.919,Z 1174.55,A -85,B 0,C 180,E1 4268.421,E2 4268.421} C_VEL
LIN {X 0,Y 227.648,Z 1182.462,A -85,B 0,C 180,E1 4262.701,E2 4262.701} C_VEL
LIN {X 0,Y 222.663,Z 1188.482,A -85,B 0,C 180,E1 4257.261,E2 4257.261} C_VEL
LIN {X 0,Y 219.192,Z 1193.378,A -85,B 0,C 180,E1 4251.685,E2 4251.685} C_VEL
LIN {X 0,Y 217.05,Z 1197.346,A -85,B 0,C 180,E1 4245.772,E2 4245.772} C_VEL
LIN {X 0,Y 216.066,Z 1200.5,A -85,B 0,C 180,E1 4239.054,E2 4239.054} C_VEL
LIN {X 0,Y 215.917,Z 1201.954,A -85,B 0,C 180,E1 4233.187,E2 4233.187} C_VEL
LIN {X 0,Y 215.914,Z 1202.35,A -85,B 0,C 180,E1 4228.143,E2 4228.143} C_VEL
LIN {X 0,Y 215.987,Z 1201.781,A -85,B 0,C 180,E1 4222.553,E2 4222.553} C_VEL
LIN {X 0,Y 216.607,Z 1199.982,A -85,B 0,C 180,E1 4216.385,E2 4216.385} C_VEL
LIN {X 0,Y 218.328,Z 1197.164,A -85,B 0,C 180,E1 4210.47,E2 4210.47} C_VEL
LIN {X 0,Y 221.617,Z 1193.137,A -85,B 0,C 180,E1 4204.471,E2 4204.471} C_VEL
LIN {X 0,Y 226.358,Z 1188.204,A -85,B 0,C 180,E1 4198.882,E2 4198.882} C_VEL
LIN {X 0,Y 232.931,Z 1182.008,A -85,B 0,C 180,E1 4193.37,E2 4193.37} C_VEL
LIN {X 0,Y 243.425,Z 1172.787,A -85,B 0,C 180,E1 4186.983,E2 4186.983} C_VEL
LIN {X 0,Y 255.229,Z 1162.406,A -85,B 0,C 180,E1 4181.562,E2 4181.562} C_VEL
LIN {X 0,Y 266.717,Z 1152.341,A -85,B 0,C 180,E1 4177.37,E2 4177.37} C_VEL
LIN {X 0,Y 278.797,Z 1141.503,A -85,B 0,C 180,E1 4173.692,E2 4173.692} C_VEL
LIN {X 0,Y 294.618,Z 1126.826,A -85,B 0,C 180,E1 4169.681,E2 4169.681} C_VEL
LIN {X 0,Y 310.941,Z 1110.481,A -85,B 0,C 180,E1 4166.214,E2 4166.214} C_VEL
LIN {X 0,Y 323.844,Z 1096.854,A -85,B 0,C 180,E1 4163.858,E2 4163.858} C_VEL
LIN {X 0,Y 336.907,Z 1082.188,A -85,B 0,C 180,E1 4161.734,E2 4161.734} C_VEL
LIN {X 0,Y 350.982,Z 1065.272,A -85,B 0,C 180,E1 4159.693,E2 4159.693} C_VEL
LIN {X 0,Y 368.001,Z 1042.84,A -85,B 0,C 180,E1 4157.509,E2 4157.509} C_VEL
LIN {X 0,Y 380.766,Z 1024.248,A -85,B 0,C 180,E1 4156.036,E2 4156.036} C_VEL
LIN {X 0,Y 392.042,Z 1006.366,A -85,B 0,C 180,E1 4154.85,E2 4154.85} C_VEL
LIN {X 0,Y 402.82,Z 987.617,A -85,B 0,C 180,E1 4153.786,E2 4153.786} C_VEL
LIN {X 0,Y 414.61,Z 964.893,A -85,B 0,C 180,E1 4152.714,E2 4152.714} C_VEL
LIN {X 0,Y 425.874,Z 939.701,A -85,B 0,C 180,E1 4151.755,E2 4151.755} C_VEL
LIN {X 0,Y 434.063,Z 918.685,A -85,B 0,C 180,E1 4151.101,E2 4151.101} C_VEL
LIN {X 0,Y 441.08,Z 897.972,A -85,B 0,C 180,E1 4150.565,E2 4150.565} C_VEL
LIN {X 0,Y 447.44,Z 875.945,A -85,B 0,C 180,E1 4150.103,E2 4150.103} C_VEL
LIN {X 0,Y 453.966,Z 847.725,A -85,B 0,C 180,E1 4149.633,E2 4149.633} C_VEL
LIN {X 0,Y 458.149,Z 822.392,A -85,B 0,C 180,E1 4149.265,E2 4149.265} C_VEL
LIN {X 0,Y 478.196,Z 647.945,A -85,B 0,C 180,E1 4146.921,E2 4146.921} C_VEL
LIN {X 0,Y 477.403,Z 644.633,A -85,B 0,C 180,E1 4142.761,E2 4142.761} C_VEL
LIN {X 0,Y 478.155,Z 648.116,A -85,B 0,C 180,E1 4138.907,E2 4138.907} C_VEL
LIN {X 0,Y 458.219,Z 821.393,A -85,B 0,C 180,E1 4136.587,E2 4136.587} C_VEL
LIN {X 0,Y 453.871,Z 847.571,A -85,B 0,C 180,E1 4136.205,E2 4136.205} C_VEL
LIN {X 0,Y 447.494,Z 874.898,A -85,B 0,C 180,E1 4135.731,E2 4135.731} C_VEL
LIN {X 0,Y 441.207,Z 896.696,A -85,B 0,C 180,E1 4135.248,E2 4135.248} C_VEL
LIN {X 0,Y 434.297,Z 917.105,A -85,B 0,C 180,E1 4134.702,E2 4134.702} C_VEL
LIN {X 0,Y 426.247,Z 937.795,A -85,B 0,C 180,E1 4134.039,E2 4134.039} C_VEL
LIN {X 0,Y 414.991,Z 963.031,A -85,B 0,C 180,E1 4133.052,E2 4133.052} C_VEL
LIN {X 0,Y 403.393,Z 985.388,A -85,B 0,C 180,E1 4131.977,E2 4131.977} C_VEL
LIN {X 0,Y 392.413,Z 1004.469,A -85,B 0,C 180,E1 4130.875,E2 4130.875} C_VEL
LIN {X 0,Y 381.806,Z 1021.291,A -85,B 0,C 180,E1 4129.742,E2 4129.742} C_VEL
LIN {X 0,Y 369.59,Z 1039.098,A -85,B 0,C 180,E1 4128.33,E2 4128.33} C_VEL
LIN {X 0,Y 353.981,Z 1059.953,A -85,B 0,C 180,E1 4126.329,E2 4126.329} C_VEL
LIN {X 0,Y 338.412,Z 1078.639,A -85,B 0,C 180,E1 4124.094,E2 4124.094} C_VEL
LIN {X 0,Y 324.835,Z 1093.822,A -85,B 0,C 180,E1 4121.887,E2 4121.887} C_VEL
LIN {X 0,Y 311.723,Z 1107.579,A -85,B 0,C 180,E1 4119.488,E2 4119.488} C_VEL
LIN {X 0,Y 296.141,Z 1123.023,A -85,B 0,C 180,E1 4116.202,E2 4116.202} C_VEL
LIN {X 0,Y 280.259,Z 1137.645,A -85,B 0,C 180,E1 4112.223,E2 4112.223} C_VEL
LIN {X 0,Y 267.608,Z 1148.82,A -85,B 0,C 180,E1 4108.416,E2 4108.416} C_VEL
LIN {X 0,Y 256.718,Z 1158.197,A -85,B 0,C 180,E1 4104.489,E2 4104.489} C_VEL
LIN {X 0,Y 245.919,Z 1167.405,A -85,B 0,C 180,E1 4099.723,E2 4099.723} C_VEL
LIN {X 0,Y 234.376,Z 1177.313,A -85,B 0,C 180,E1 4093.044,E2 4093.044} C_VEL
LIN {X 0,Y 227.286,Z 1183.668,A -85,B 0,C 180,E1 4087.378,E2 4087.378} C_VEL
LIN {X 0,Y 222.264,Z 1188.58,A -85,B 0,C 180,E1 4081.757,E2 4081.757} C_VEL
LIN {X 0,Y 218.883,Z 1192.392,A -85,B 0,C 180,E1 4076.009,E2 4076.009} C_VEL
LIN {X 0,Y 216.938,Z 1195.14,A -85,B 0,C 180,E1 4070.222,E2 4070.222} C_VEL
LIN {X 0,Y 216.119,Z 1196.853,A -85,B 0,C 180,E1 4064.466,E2 4064.466} C_VEL
LIN {X 0,Y 215.934,Z 1197.533,A -85,B 0,C 180,E1 4059.057,E2 4059.057} C_VEL
LIN {X 0,Y 215.919,Z 1197.334,A -85,B 0,C 180,E1 4053.982,E2 4053.982} C_VEL
LIN {X 0,Y 216.023,Z 1196.336,A -85,B 0,C 180,E1 4048.938,E2 4048.938} C_VEL
LIN {X 0,Y 216.499,Z 1194.432,A -85,B 0,C 180,E1 4043.635,E2 4043.635} C_VEL
LIN {X 0,Y 217.872,Z 1191.48,A -85,B 0,C 180,E1 4038.081,E2 4038.081} C_VEL
LIN {X 0,Y 221.244,Z 1186.517,A -85,B 0,C 180,E1 4031.283,E2 4031.283} C_VEL
LIN {X 0,Y 226.961,Z 1179.486,A -85,B 0,C 180,E1 4024.421,E2 4024.421} C_VEL
LIN {X 0,Y 233.415,Z 1172.503,A -85,B 0,C 180,E1 4019.066,E2 4019.066} C_VEL
LIN {X 0,Y 241.062,Z 1164.679,A -85,B 0,C 180,E1 4014.207,E2 4014.207} C_VEL
LIN {X 0,Y 251.508,Z 1154.313,A -85,B 0,C 180,E1 4009.006,E2 4009.006} C_VEL
LIN {X 0,Y 264.705,Z 1141.023,A -85,B 0,C 180,E1 4003.823,E2 4003.823} C_VEL
LIN {X 0,Y 276.278,Z 1129.122,A -85,B 0,C 180,E1 4000.107,E2 4000.107} C_VEL
LIN {X 0,Y 287.763,Z 1116.906,A -85,B 0,C 180,E1 3996.948,E2 3996.948} C_VEL
LIN {X 0,Y 300.892,Z 1102.313,A -85,B 0,C 180,E1 3993.822,E2 3993.822} C_VEL
LIN {X 0,Y 316.943,Z 1083.191,A -85,B 0,C 180,E1 3990.542,E2 3990.542} C_VEL
LIN {X 0,Y 329.368,Z 1067.254,A -85,B 0,C 180,E1 3988.312,E2 3988.312} C_VEL
LIN {X 0,Y 341.082,Z 1051.183,A -85,B 0,C 180,E1 3986.417,E2 3986.417} C_VEL
LIN {X 0,Y 353.136,Z 1033.38,A -85,B 0,C 180,E1 3984.647,E2 3984.647} C_VEL
LIN {X 0,Y 367.629,Z 1009.831,A -85,B 0,C 180,E1 3982.719,E2 3982.719} C_VEL
LIN {X 0,Y 378.956,Z 989.219,A -85,B 0,C 180,E1 3981.346,E2 3981.346} C_VEL
LIN {X 0,Y 388.485,Z 970.037,A -85,B 0,C 180,E1 3980.257,E2 3980.257} C_VEL
LIN {X 0,Y 397.313,Z 950.335,A -85,B 0,C 180,E1 3979.312,E2 3979.312} C_VEL
LIN {X 0,Y 407.215,Z 925.398,A -85,B 0,C 180,E1 3978.318,E2 3978.318} C_VEL
LIN {X 0,Y 415.705,Z 899.6,A -85,B 0,C 180,E1 3977.497,E2 3977.497} C_VEL
LIN {X 0,Y 421.659,Z 878.284,A -85,B 0,C 180,E1 3976.948,E2 3976.948} C_VEL
LIN {X 0,Y 426.647,Z 856.878,A -85,B 0,C 180,E1 3976.5,E2 3976.5} C_VEL
LIN {X 0,Y 431.224,Z 832.037,A -85,B 0,C 180,E1 3976.078,E2 3976.078} C_VEL
LIN {X 0,Y 435.591,Z 795.582,A -85,B 0,C 180,E1 3975.539,E2 3975.539} C_VEL
LIN {X 0,Y 449.631,Z 660.025,A -85,B 0,C 180,E1 3973.631,E2 3973.631} C_VEL
LIN {X 0,Y 449.973,Z 655.035,A -85,B 0,C 180,E1 3973.435,E2 3973.435} C_VEL
LIN {X 0,Y 450.224,Z 642.663,A -85,B 0,C 180,E1 3972.48,E2 3972.48} C_VEL
LIN {X 0,Y 450.56,Z 638.357,A -85,B 0,C 180,E1 3972.323,E2 3972.323} C_VEL
LIN {X 0,Y 451.054,Z 633.696,A -85,B 0,C 180,E1 3972.255,E2 3972.255} C_VEL
LIN {X 0,Y 449.491,Z 630.36,A -85,B 0,C 180,E1 3970.51,E2 3970.51} C_VEL
LIN {X 0,Y 448.174,Z 627.428,A -85,B 0,C 180,E1 3968.597,E2 3968.597} C_VEL
LIN {X 0,Y 446.822,Z 623.647,A -85,B 0,C 180,E1 3965.007,E2 3965.007} C_VEL
LIN {X 0,Y 446.864,Z 623.755,A -85,B 0,C 180,E1 3960.897,E2 3960.897} C_VEL
LIN {X 0,Y 448.656,Z 628.486,A -85,B 0,C 180,E1 3956.742,E2 3956.742} C_VEL
LIN {X 0,Y 450.644,Z 632.842,A -85,B 0,C 180,E1 3954.27,E2 3954.27} C_VEL
LIN {X 0,Y 451.064,Z 634.025,A -85,B 0,C 180,E1 3953.81,E2 3953.81} C_VEL
LIN {X 0,Y 430.923,Z 822.727,A -85,B 0,C 180,E1 3951.177,E2 3951.177} C_VEL
LIN {X 0,Y 426.935,Z 848.176,A -85,B 0,C 180,E1 3950.78,E2 3950.78} C_VEL
LIN {X 0,Y 420.667,Z 876.384,A -85,B 0,C 180,E1 3950.263,E2 3950.263} C_VEL
LIN {X 0,Y 414.572,Z 898.406,A -85,B 0,C 180,E1 3949.747,E2 3949.747} C_VEL
LIN {X 0,Y 407.955,Z 918.817,A -85,B 0,C 180,E1 3949.162,E2 3949.162} C_VEL
LIN {X 0,Y 400.076,Z 939.968,A -85,B 0,C 180,E1 3948.435,E2 3948.435} C_VEL
LIN {X 0,Y 388.916,Z 966.007,A -85,B 0,C 180,E1 3947.336,E2 3947.336} C_VEL
LIN {X 0,Y 377.902,Z 988.248,A -85,B 0,C 180,E1 3946.177,E2 3946.177} C_VEL
LIN {X 0,Y 367.493,Z 1007.24,A -85,B 0,C 180,E1 3944.992,E2 3944.992} C_VEL
LIN {X 0,Y 356.826,Z 1025.024,A -85,B 0,C 180,E1 3943.686,E2 3943.686} C_VEL
LIN {X 0,Y 343.045,Z 1046.104,A -85,B 0,C 180,E1 3941.842,E2 3941.842} C_VEL
LIN {X 0,Y 328.032,Z 1066.716,A -85,B 0,C 180,E1 3939.603,E2 3939.603} C_VEL
LIN {X 0,Y 315.478,Z 1082.693,A -85,B 0,C 180,E1 3937.501,E2 3937.501} C_VEL
LIN {X 0,Y 303.006,Z 1097.595,A -85,B 0,C 180,E1 3935.158,E2 3935.158} C_VEL
LIN {X 0,Y 288.6,Z 1113.842,A -85,B 0,C 180,E1 3932.065,E2 3932.065} C_VEL
LIN {X 0,Y 273.125,Z 1130.14,A -85,B 0,C 180,E1 3928.139,E2 3928.139} C_VEL
LIN {X 0,Y 261.322,Z 1142.031,A -85,B 0,C 180,E1 3924.587,E2 3924.587} C_VEL
LIN {X 0,Y 250.536,Z 1152.639,A -85,B 0,C 180,E1 3920.738,E2 3920.738} C_VEL
LIN {X 0,Y 239.895,Z 1162.992,A -85,B 0,C 180,E1 3916.143,E2 3916.143} C_VEL
LIN {X 0,Y 228.389,Z 1174.324,A -85,B 0,C 180,E1 3909.732,E2 3909.732} C_VEL
LIN {X 0,Y 220.648,Z 1182.257,A -85,B 0,C 180,E1 3903.876,E2 3903.876} C_VEL
LIN {X 0,Y 215.3,Z 1188.298,A -85,B 0,C 180,E1 3898.276,E2 3898.276} C_VEL
LIN {X 0,Y 211.678,Z 1193.001,A -85,B 0,C 180,E1 3892.79,E2 3892.79} C_VEL
LIN {X 0,Y 209.424,Z 1196.709,A -85,B 0,C 180,E1 3887.219,E2 3887.219} C_VEL
LIN {X 0,Y 208.285,Z 1199.447,A -85,B 0,C 180,E1 3881.633,E2 3881.633} C_VEL
LIN {X 0,Y 207.961,Z 1201.097,A -85,B 0,C 180,E1 3876.627,E2 3876.627} C_VEL
LIN {X 0,Y 207.917,Z 1201.973,A -85,B 0,C 180,E1 3871.93,E2 3871.93} C_VEL
LIN {X 0,Y 207.916,Z 1202.176,A -85,B 0,C 180,E1 3866.969,E2 3866.969} C_VEL
LIN {X 0,Y 208.041,Z 1201.508,A -85,B 0,C 180,E1 3861.433,E2 3861.433} C_VEL
LIN {X 0,Y 208.816,Z 1199.703,A -85,B 0,C 180,E1 3855.298,E2 3855.298} C_VEL
LIN {X 0,Y 210.715,Z 1196.971,A -85,B 0,C 180,E1 3849.444,E2 3849.444} C_VEL
LIN {X 0,Y 214.259,Z 1193.024,A -85,B 0,C 180,E1 3843.386,E2 3843.386} C_VEL
LIN {X 0,Y 219.263,Z 1188.208,A -85,B 0,C 180,E1 3837.756,E2 3837.756} C_VEL
LIN {X 0,Y 226.268,Z 1182.03,A -85,B 0,C 180,E1 3832.105,E2 3832.105} C_VEL
LIN {X 0,Y 236.861,Z 1173.253,A -85,B 0,C 180,E1 3825.853,E2 3825.853} C_VEL
LIN {X 0,Y 249.748,Z 1162.491,A -85,B 0,C 180,E1 3820.123,E2 3820.123} C_VEL
LIN {X 0,Y 261.718,Z 1152.449,A -85,B 0,C 180,E1 3815.912,E2 3815.912} C_VEL
LIN {X 0,Y 274.246,Z 1141.636,A -85,B 0,C 180,E1 3812.239,E2 3812.239} C_VEL
LIN {X 0,Y 289.869,Z 1127.617,A -85,B 0,C 180,E1 3808.408,E2 3808.408} C_VEL
LIN {X 0,Y 306.612,Z 1111.456,A -85,B 0,C 180,E1 3804.966,E2 3804.966} C_VEL
LIN {X 0,Y 320.419,Z 1097.274,A -85,B 0,C 180,E1 3802.533,E2 3802.533} C_VEL
LIN {X 0,Y 333.136,Z 1083.377,A -85,B 0,C 180,E1 3800.541,E2 3800.541} C_VEL
LIN {X 0,Y 346.223,Z 1068.083,A -85,B 0,C 180,E1 3798.696,E2 3798.696} C_VEL
LIN {X 0,Y 359.935,Z 1050.826,A -85,B 0,C 180,E1 3796.959,E2 3796.959} C_VEL
LIN {X 0,Y 376.452,Z 1027.946,A -85,B 0,C 180,E1 3795.088,E2 3795.088} C_VEL
LIN {X 0,Y 389.165,Z 1008.312,A -85,B 0,C 180,E1 3793.79,E2 3793.79} C_VEL
LIN {X 0,Y 399.84,Z 990.203,A -85,B 0,C 180,E1 3792.773,E2 3792.773} C_VEL
LIN {X 0,Y 410.197,Z 970.835,A -85,B 0,C 180,E1 3791.857,E2 3791.857} C_VEL
LIN {X 0,Y 420.661,Z 948.958,A -85,B 0,C 180,E1 3790.992,E2 3790.992} C_VEL
LIN {X 0,Y 431.682,Z 922.136,A -85,B 0,C 180,E1 3790.138,E2 3790.138} C_VEL
LIN {X 0,Y 439.327,Z 900.206,A -85,B 0,C 180,E1 3789.576,E2 3789.576} C_VEL
LIN {X 0,Y 445.653,Z 878.928,A -85,B 0,C 180,E1 3789.133,E2 3789.133} C_VEL
LIN {X 0,Y 451.169,Z 856.567,A -85,B 0,C 180,E1 3788.759,E2 3788.759} C_VEL
LIN {X 0,Y 456.535,Z 828.074,A -85,B 0,C 180,E1 3788.342,E2 3788.342} C_VEL
LIN {X 0,Y 462.401,Z 780.011,A -85,B 0,C 180,E1 3787.699,E2 3787.699} C_VEL
LIN {X 0,Y 476.831,Z 655.285,A -85,B 0,C 180,E1 3786.05,E2 3786.05} C_VEL
LIN {X 0,Y 476.42,Z 652.623,A -85,B 0,C 180,E1 3782.767,E2 3782.767} C_VEL
LIN {X 0,Y 476.8,Z 655.427,A -85,B 0,C 180,E1 3779.773,E2 3779.773} C_VEL
LIN {X 0,Y 457.362,Z 821.607,A -85,B 0,C 180,E1 3777.584,E2 3777.584} C_VEL
LIN {X 0,Y 452.851,Z 848.358,A -85,B 0,C 180,E1 3777.203,E2 3777.203} C_VEL
LIN {X 0,Y 446.409,Z 875.443,A -85,B 0,C 180,E1 3776.746,E2 3776.746} C_VEL
LIN {X 0,Y 440.116,Z 896.98,A -85,B 0,C 180,E1 3776.283,E2 3776.283} C_VEL
LIN {X 0,Y 433.129,Z 917.363,A -85,B 0,C 180,E1 3775.755,E2 3775.755} C_VEL
LIN {X 0,Y 425.035,Z 937.913,A -85,B 0,C 180,E1 3775.117,E2 3775.117} C_VEL
LIN {X 0,Y 413.593,Z 963.232,A -85,B 0,C 180,E1 3774.157,E2 3774.157} C_VEL
LIN {X 0,Y 401.842,Z 985.577,A -85,B 0,C 180,E1 3773.116,E2 3773.116} C_VEL
LIN {X 0,Y 390.707,Z 1004.646,A -85,B 0,C 180,E1 3772.045,E2 3772.045} C_VEL
LIN {X 0,Y 379.555,Z 1022.025,A -85,B 0,C 180,E1 3770.905,E2 3770.905} C_VEL
LIN {X 0,Y 366.182,Z 1041.111,A -85,B 0,C 180,E1 3769.415,E2 3769.415} C_VEL
LIN {X 0,Y 349.448,Z 1062.676,A -85,B 0,C 180,E1 3767.34,E2 3767.34} C_VEL
LIN {X 0,Y 334.763,Z 1079.863,A -85,B 0,C 180,E1 3765.292,E2 3765.292} C_VEL
LIN {X 0,Y 321.627,Z 1094.184,A -85,B 0,C 180,E1 3763.235,E2 3763.235} C_VEL
LIN {X 0,Y 308.018,Z 1108.089,A -85,B 0,C 180,E1 3760.842,E2 3760.842} C_VEL
LIN {X 0,Y 291.274,Z 1124.176,A -85,B 0,C 180,E1 3757.428,E2 3757.428} C_VEL
LIN {X 0,Y 275.631,Z 1138.043,A -85,B 0,C 180,E1 3753.637,E2 3753.637} C_VEL
LIN {X 0,Y 263.157,Z 1148.66,A -85,B 0,C 180,E1 3750.029,E2 3750.029} C_VEL
LIN {X 0,Y 251.761,Z 1158.063,A -85,B 0,C 180,E1 3746.102,E2 3746.102} C_VEL
LIN {X 0,Y 240.553,Z 1167.152,A -85,B 0,C 180,E1 3741.391,E2 3741.391} C_VEL
LIN {X 0,Y 228.511,Z 1176.948,A -85,B 0,C 180,E1 3734.785,E2 3734.785} C_VEL
LIN {X 0,Y 220.5,Z 1183.635,A -85,B 0,C 180,E1 3728.738,E2 3728.738} C_VEL
LIN {X 0,Y 215.039,Z 1188.569,A -85,B 0,C 180,E1 3722.956,E2 3722.956} C_VEL
LIN {X 0,Y 211.304,Z 1192.405,A -85,B 0,C 180,E1 3717.016,E2 3717.016} C_VEL
LIN {X 0,Y 209.161,Z 1195.094,A -85,B 0,C 180,E1 3711.22,E2 3711.22} C_VEL
LIN {X 0,Y 208.219,Z 1196.776,A -85,B 0,C 180,E1 3705.598,E2 3705.598} C_VEL
LIN {X 0,Y 207.951,Z 1197.523,A -85,B 0,C 180,E1 3700.527,E2 3700.527} C_VEL
LIN {X 0,Y 207.913,Z 1197.593,A -85,B 0,C 180,E1 3696.072,E2 3696.072} C_VEL
LIN {X 0,Y 207.955,Z 1196.927,A -85,B 0,C 180,E1 3690.825,E2 3690.825} C_VEL
LIN {X 0,Y 208.278,Z 1195.355,A -85,B 0,C 180,E1 3685.318,E2 3685.318} C_VEL
LIN {X 0,Y 209.478,Z 1192.583,A -85,B 0,C 180,E1 3679.271,E2 3679.271} C_VEL
LIN {X 0,Y 211.821,Z 1188.928,A -85,B 0,C 180,E1 3673.546,E2 3673.546} C_VEL
LIN {X 0,Y 215.548,Z 1184.255,A -85,B 0,C 180,E1 3667.929,E2 3667.929} C_VEL
LIN {X 0,Y 220.774,Z 1178.534,A -85,B 0,C 180,E1 3662.486,E2 3662.486} C_VEL
LIN {X 0,Y 227.887,Z 1171.378,A -85,B 0,C 180,E1 3657.038,E2 3657.038} C_VEL
LIN {X 0,Y 238.942,Z 1160.784,A -85,B 0,C 180,E1 3650.729,E2 3650.729} C_VEL
LIN {X 0,Y 250.465,Z 1149.731,A -85,B 0,C 180,E1 3645.683,E2 3645.683} C_VEL
LIN {X 0,Y 261.403,Z 1139.136,A -85,B 0,C 180,E1 3641.764,E2 3641.764} C_VEL
LIN {X 0,Y 273.365,Z 1127.23,A -85,B 0,C 180,E1 3638.149,E2 3638.149} C_VEL
LIN {X 0,Y 288.255,Z 1111.803,A -85,B 0,C 180,E1 3634.354,E2 3634.354} C_VEL
LIN {X 0,Y 303.472,Z 1094.753,A -85,B 0,C 180,E1 3631.057,E2 3631.057} C_VEL
LIN {X 0,Y 315.846,Z 1080.078,A -85,B 0,C 180,E1 3628.728,E2 3628.728} C_VEL
LIN {X 0,Y 327.911,Z 1064.824,A -85,B 0,C 180,E1 3626.692,E2 3626.692} C_VEL
LIN {X 0,Y 341.525,Z 1046.33,A -85,B 0,C 180,E1 3624.625,E2 3624.625} C_VEL
LIN {X 0,Y 356.33,Z 1024.048,A -85,B 0,C 180,E1 3622.602,E2 3622.602} C_VEL
LIN {X 0,Y 367.369,Z 1005.75,A -85,B 0,C 180,E1 3621.223,E2 3621.223} C_VEL
LIN {X 0,Y 377.795,Z 986.845,A -85,B 0,C 180,E1 3620.023,E2 3620.023} C_VEL
LIN {X 0,Y 387.414,Z 967.563,A -85,B 0,C 180,E1 3618.978,E2 3618.978} C_VEL
LIN {X 0,Y 398.208,Z 943.376,A -85,B 0,C 180,E1 3617.889,E2 3617.889} C_VEL
LIN {X 0,Y 407.279,Z 919.396,A -85,B 0,C 180,E1 3617.014,E2 3617.014} C_VEL
LIN {X 0,Y 414.258,Z 898.119,A -85,B 0,C 180,E1 3616.376,E2 3616.376} C_VEL
LIN {X 0,Y 420.154,Z 877.068,A -85,B 0,C 180,E1 3615.854,E2 3615.854} C_VEL
LIN {X 0,Y 425.319,Z 854.875,A -85,B 0,C 180,E1 3615.409,E2 3615.409} C_VEL
LIN {X 0,Y 430.389,Z 826.193,A -85,B 0,C 180,E1 3614.944,E2 3614.944} C_VEL
LIN {X 0,Y 435.819,Z 777.648,A -85,B 0,C 180,E1 3614.253,E2 3614.253} C_VEL
LIN {X 0,Y 450.56,Z 638.357,A -85,B 0,C 180,E1 3612.323,E2 3612.323} C_VEL
LIN {X 0,Y 450.599,Z 636.403,A -85,B 0,C 180,E1 3612.16,E2 3612.16} C_VEL
LIN {X 0,Y 450.291,Z 635.167,A -85,B 0,C 180,E1 3611.781,E2 3611.781} C_VEL
LIN {X 0,Y 449.571,Z 635.091,A -85,B 0,C 180,E1 3611.144,E2 3611.144} C_VEL
LIN {X 0,Y 447.973,Z 636.787,A -85,B 0,C 180,E1 3609.756,E2 3609.756} C_VEL
LIN {X 0,Y 447.612,Z 636.456,A -85,B 0,C 180,E1 3609.294,E2 3609.294} C_VEL
LIN {X 0,Y 446.963,Z 635.084,A -85,B 0,C 180,E1 3608.232,E2 3608.232} C_VEL
LIN {X 0,Y 445.817,Z 631.573,A -85,B 0,C 180,E1 3604.889,E2 3604.889} C_VEL
LIN {X 0,Y 445.873,Z 631.8,A -85,B 0,C 180,E1 3600.899,E2 3600.899} C_VEL
LIN {X 0,Y 447.539,Z 636.279,A -85,B 0,C 180,E1 3596.926,E2 3596.926} C_VEL
LIN {X 0,Y 449.204,Z 640.033,A -85,B 0,C 180,E1 3594.74,E2 3594.74} C_VEL
LIN {X 0,Y 429.369,Z 822.642,A -85,B 0,C 180,E1 3592.227,E2 3592.227} C_VEL
LIN {X 0,Y 425.322,Z 848.123,A -85,B 0,C 180,E1 3591.837,E2 3591.837} C_VEL
LIN {X 0,Y 418.987,Z 876.311,A -85,B 0,C 180,E1 3591.336,E2 3591.336} C_VEL
LIN {X 0,Y 412.96,Z 897.878,A -85,B 0,C 180,E1 3590.847,E2 3590.847} C_VEL
LIN {X 0,Y 406.122,Z 918.746,A -85,B 0,C 180,E1 3590.268,E2 3590.268} C_VEL
LIN {X 0,Y 398.447,Z 939.122,A -85,B 0,C 180,E1 3589.59,E2 3589.59} C_VEL
LIN {X 0,Y 387.639,Z 964.275,A -85,B 0,C 180,E1 3588.573,E2 3588.573} C_VEL
LIN {X 0,Y 376.007,Z 987.503,A -85,B 0,C 180,E1 3587.404,E2 3587.404} C_VEL
LIN {X 0,Y 365.431,Z 1006.558,A -85,B 0,C 180,E1 3586.25,E2 3586.25} C_VEL
LIN {X 0,Y 355.002,Z 1023.716,A -85,B 0,C 180,E1 3585.034,E2 3585.034} C_VEL
LIN {X 0,Y 343.049,Z 1041.794,A -85,B 0,C 180,E1 3583.524,E2 3583.524} C_VEL
LIN {X 0,Y 327.653,Z 1063.109,A -85,B 0,C 180,E1 3581.359,E2 3581.359} C_VEL
LIN {X 0,Y 312.751,Z 1081.759,A -85,B 0,C 180,E1 3578.994,E2 3578.994} C_VEL
LIN {X 0,Y 300.328,Z 1096.304,A -85,B 0,C 180,E1 3576.764,E2 3576.764} C_VEL
LIN {X 0,Y 287.647,Z 1110.292,A -85,B 0,C 180,E1 3574.198,E2 3574.198} C_VEL
LIN {X 0,Y 272.814,Z 1125.797,A -85,B 0,C 180,E1 3570.726,E2 3570.726} C_VEL
LIN {X 0,Y 257.754,Z 1140.542,A -85,B 0,C 180,E1 3566.516,E2 3566.516} C_VEL
LIN {X 0,Y 245.827,Z 1151.818,A -85,B 0,C 180,E1 3562.481,E2 3562.481} C_VEL
LIN {X 0,Y 235.116,Z 1161.781,A -85,B 0,C 180,E1 3558.093,E2 3558.093} C_VEL
LIN {X 0,Y 224.871,Z 1171.343,A -85,B 0,C 180,E1 3552.869,E2 3552.869} C_VEL
LIN {X 0,Y 214.378,Z 1181.43,A -85,B 0,C 180,E1 3545.664,E2 3545.664} C_VEL
LIN {X 0,Y 208.231,Z 1187.852,A -85,B 0,C 180,E1 3539.642,E2 3539.642} C_VEL
LIN {X 0,Y 204.248,Z 1192.623,A -85,B 0,C 180,E1 3533.975,E2 3533.975} C_VEL
LIN {X 0,Y 201.7,Z 1196.398,A -85,B 0,C 180,E1 3528.199,E2 3528.199} C_VEL
LIN {X 0,Y 200.412,Z 1199.085,A -85,B 0,C 180,E1 3522.682,E2 3522.682} C_VEL
LIN {X 0,Y 199.987,Z 1200.846,A -85,B 0,C 180,E1 3517.47,E2 3517.47} C_VEL
LIN {X 0,Y 199.916,Z 1201.854,A -85,B 0,C 180,E1 3512.294,E2 3512.294} C_VEL
LIN {X 0,Y 199.915,Z 1202.12,A -85,B 0,C 180,E1 3507.134,E2 3507.134} C_VEL
LIN {X 0,Y 200.058,Z 1201.444,A -85,B 0,C 180,E1 3501.088,E2 3501.088} C_VEL
LIN {X 0,Y 200.935,Z 1199.655,A -85,B 0,C 180,E1 3494.709,E2 3494.709} C_VEL
LIN {X 0,Y 203.17,Z 1196.779,A -85,B 0,C 180,E1 3488.341,E2 3488.341} C_VEL
LIN {X 0,Y 207.091,Z 1192.803,A -85,B 0,C 180,E1 3482.075,E2 3482.075} C_VEL
LIN {X 0,Y 212.853,Z 1187.703,A -85,B 0,C 180,E1 3476.015,E2 3476.015} C_VEL
LIN {X 0,Y 221.286,Z 1180.844,A -85,B 0,C 180,E1 3469.75,E2 3469.75} C_VEL
LIN {X 0,Y 233.821,Z 1170.939,A -85,B 0,C 180,E1 3463.011,E2 3463.011} C_VEL
LIN {X 0,Y 245.569,Z 1161.667,A -85,B 0,C 180,E1 3458.204,E2 3458.204} C_VEL
LIN {X 0,Y 257.511,Z 1152.048,A -85,B 0,C 180,E1 3454.205,E2 3454.205} C_VEL
LIN {X 0,Y 270.55,Z 1141.201,A -85,B 0,C 180,E1 3450.562,E2 3450.562} C_VEL
LIN {X 0,Y 287.446,Z 1126.509,A -85,B 0,C 180,E1 3446.626,E2 3446.626} C_VEL
LIN {X 0,Y 304.739,Z 1110.147,A -85,B 0,C 180,E1 3443.265,E2 3443.265} C_VEL
LIN {X 0,Y 318.94,Z 1095.852,A -85,B 0,C 180,E1 3440.899,E2 3440.899} C_VEL
LIN {X 0,Y 332.816,Z 1080.915,A -85,B 0,C 180,E1 3438.856,E2 3438.856} C_VEL
LIN {X 0,Y 349.217,Z 1061.896,A -85,B 0,C 180,E1 3436.72,E2 3436.72} C_VEL
LIN {X 0,Y 365.179,Z 1041.234,A -85,B 0,C 180,E1 3434.869,E2 3434.869} C_VEL
LIN {X 0,Y 377.494,Z 1023.824,A -85,B 0,C 180,E1 3433.574,E2 3433.574} C_VEL
LIN {X 0,Y 389.112,Z 1005.919,A -85,B 0,C 180,E1 3432.46,E2 3432.46} C_VEL
LIN {X 0,Y 399.955,Z 987.569,A -85,B 0,C 180,E1 3431.485,E2 3431.485} C_VEL
LIN {X 0,Y 412.255,Z 964.464,A -85,B 0,C 180,E1 3430.467,E2 3430.467} C_VEL
LIN {X 0,Y 423.84,Z 939.091,A -85,B 0,C 180,E1 3429.569,E2 3429.569} C_VEL
LIN {X 0,Y 432.217,Z 918.011,A -85,B 0,C 180,E1 3428.961,E2 3428.961} C_VEL
LIN {X 0,Y 439.44,Z 897.059,A -85,B 0,C 180,E1 3428.462,E2 3428.462} C_VEL
LIN {X 0,Y 446.177,Z 874.03,A -85,B 0,C 180,E1 3428.018,E2 3428.018} C_VEL
LIN {X 0,Y 452.914,Z 844.511,A -85,B 0,C 180,E1 3427.567,E2 3427.567} C_VEL
LIN {X 0,Y 456.788,Z 821.167,A -85,B 0,C 180,E1 3427.244,E2 3427.244} C_VEL
LIN {X 0,Y 475.588,Z 662.567,A -85,B 0,C 180,E1 3425.187,E2 3425.187} C_VEL
LIN {X 0,Y 475.438,Z 660.612,A -85,B 0,C 180,E1 3422.773,E2 3422.773} C_VEL
LIN {X 0,Y 475.572,Z 662.588,A -85,B 0,C 180,E1 3420.647,E2 3420.647} C_VEL
LIN {X 0,Y 456.68,Z 821.624,A -85,B 0,C 180,E1 3418.588,E2 3418.588} C_VEL
LIN {X 0,Y 452.182,Z 848.02,A -85,B 0,C 180,E1 3418.222,E2 3418.222} C_VEL
LIN {X 0,Y 445.65,Z 875.328,A -85,B 0,C 180,E1 3417.777,E2 3417.777} C_VEL
LIN {X 0,Y 439.169,Z 897.265,A -85,B 0,C 180,E1 3417.323,E2 3417.323} C_VEL
LIN {X 0,Y 432.162,Z 917.478,A -85,B 0,C 180,E1 3416.817,E2 3416.817} C_VEL
LIN {X 0,Y 423.878,Z 938.263,A -85,B 0,C 180,E1 3416.193,E2 3416.193} C_VEL
LIN {X 0,Y 412.348,Z 963.435,A -85,B 0,C 180,E1 3415.27,E2 3415.27} C_VEL
LIN {X 0,Y 400.526,Z 985.635,A -85,B 0,C 180,E1 3414.269,E2 3414.269} C_VEL
LIN {X 0,Y 389.632,Z 1004.072,A -85,B 0,C 180,E1 3413.269,E2 3413.269} C_VEL
LIN {X 0,Y 378.463,Z 1021.285,A -85,B 0,C 180,E1 3412.186,E2 3412.186} C_VEL
LIN {X 0,Y 366.202,Z 1038.618,A -85,B 0,C 180,E1 3410.888,E2 3410.888} C_VEL
LIN {X 0,Y 352.127,Z 1056.882,A -85,B 0,C 180,E1 3409.254,E2 3409.254} C_VEL
LIN {X 0,Y 334.561,Z 1077.48,A -85,B 0,C 180,E1 3406.976,E2 3406.976} C_VEL
LIN {X 0,Y 320.088,Z 1093.014,A -85,B 0,C 180,E1 3404.845,E2 3404.845} C_VEL
LIN {X 0,Y 306.025,Z 1107.094,A -85,B 0,C 180,E1 3402.506,E2 3402.506} C_VEL
LIN {X 0,Y 291.106,Z 1121.102,A -85,B 0,C 180,E1 3399.664,E2 3399.664} C_VEL
LIN {X 0,Y 272.596,Z 1137.273,A -85,B 0,C 180,E1 3395.456,E2 3395.456} C_VEL
LIN {X 0,Y 258.624,Z 1148.742,A -85,B 0,C 180,E1 3391.605,E2 3391.605} C_VEL
LIN {X 0,Y 246.416,Z 1158.398,A -85,B 0,C 180,E1 3387.562,E2 3387.562} C_VEL
LIN {X 0,Y 234.179,Z 1167.867,A -85,B 0,C 180,E1 3382.575,E2 3382.575} C_VEL
LIN {X 0,Y 221.604,Z 1177.505,A -85,B 0,C 180,E1 3375.839,E2 3375.839} C_VEL
LIN {X 0,Y 213.36,Z 1183.981,A -85,B 0,C 180,E1 3369.774,E2 3369.774} C_VEL
LIN {X 0,Y 207.669,Z 1188.768,A -85,B 0,C 180,E1 3363.952,E2 3363.952} C_VEL
LIN {X 0,Y 203.634,Z 1192.578,A -85,B 0,C 180,E1 3357.804,E2 3357.804} C_VEL
LIN {X 0,Y 201.237,Z 1195.323,A -85,B 0,C 180,E1 3351.571,E2 3351.571} C_VEL
LIN {X 0,Y 200.193,Z 1197.034,A -85,B 0,C 180,E1 3345.349,E2 3345.349} C_VEL
LIN {X 0,Y 199.938,Z 1197.71,A -85,B 0,C 180,E1 3339.498,E2 3339.498} C_VEL
LIN {X 0,Y 199.917,Z 1197.531,A -85,B 0,C 180,E1 3334.301,E2 3334.301} C_VEL
LIN {X 0,Y 200.007,Z 1196.71,A -85,B 0,C 180,E1 3329.426,E2 3329.426} C_VEL
LIN {X 0,Y 200.401,Z 1195.161,A -85,B 0,C 180,E1 3324.272,E2 3324.272} C_VEL
LIN {X 0,Y 201.665,Z 1192.59,A -85,B 0,C 180,E1 3318.56,E2 3318.56} C_VEL
LIN {X 0,Y 204.243,Z 1188.912,A -85,B 0,C 180,E1 3312.624,E2 3312.624} C_VEL
LIN {X 0,Y 208.293,Z 1184.215,A -85,B 0,C 180,E1 3306.818,E2 3306.818} C_VEL
LIN {X 0,Y 213.901,Z 1178.469,A -85,B 0,C 180,E1 3301.217,E2 3301.217} C_VEL
LIN {X 0,Y 221.869,Z 1170.943,A -85,B 0,C 180,E1 3295.4,E2 3295.4} C_VEL
LIN {X 0,Y 234.38,Z 1159.491,A -85,B 0,C 180,E1 3288.663,E2 3288.663} C_VEL
LIN {X 0,Y 245.233,Z 1149.557,A -85,B 0,C 180,E1 3284.143,E2 3284.143} C_VEL
LIN {X 0,Y 256.634,Z 1138.932,A -85,B 0,C 180,E1 3280.213,E2 3280.213} C_VEL
LIN {X 0,Y 269.05,Z 1126.991,A -85,B 0,C 180,E1 3276.608,E2 3276.608} C_VEL
LIN {X 0,Y 285.118,Z 1110.738,A -85,B 0,C 180,E1 3272.684,E2 3272.684} C_VEL
LIN {X 0,Y 299.366,Z 1095.229,A -85,B 0,C 180,E1 3269.726,E2 3269.726} C_VEL
LIN {X 0,Y 312.035,Z 1080.587,A -85,B 0,C 180,E1 3267.424,E2 3267.424} C_VEL
LIN {X 0,Y 324.364,Z 1065.368,A -85,B 0,C 180,E1 3265.418,E2 3265.418} C_VEL
LIN {X 0,Y 337.544,Z 1047.867,A -85,B 0,C 180,E1 3263.482,E2 3263.482} C_VEL
LIN {X 0,Y 353.327,Z 1024.731,A -85,B 0,C 180,E1 3261.402,E2 3261.402} C_VEL
LIN {X 0,Y 364.976,Z 1005.756,A -85,B 0,C 180,E1 3260.002,E2 3260.002} C_VEL
LIN {X 0,Y 375.562,Z 986.849,A -85,B 0,C 180,E1 3258.832,E2 3258.832} C_VEL
LIN {X 0,Y 385.85,Z 966.492,A -85,B 0,C 180,E1 3257.762,E2 3257.762} C_VEL
LIN {X 0,Y 397.868,Z 939.293,A -85,B 0,C 180,E1 3256.601,E2 3256.601} C_VEL
LIN {X 0,Y 406.093,Z 917.571,A -85,B 0,C 180,E1 3255.848,E2 3255.848} C_VEL
LIN {X 0,Y 412.728,Z 897.426,A -85,B 0,C 180,E1 3255.268,E2 3255.268} C_VEL
LIN {X 0,Y 418.691,Z 876.257,A -85,B 0,C 180,E1 3254.762,E2 3254.762} C_VEL
LIN {X 0,Y 424.283,Z 852.213,A -85,B 0,C 180,E1 3254.301,E2 3254.301} C_VEL
LIN {X 0,Y 429.213,Z 823.176,A -85,B 0,C 180,E1 3253.851,E2 3253.851} C_VEL
LIN {X 0,Y 436.877,Z 753.929,A -85,B 0,C 180,E1 3252.888,E2 3252.888} C_VEL
LIN {X 0,Y 449.164,Z 639.913,A -85,B 0,C 180,E1 3251.316,E2 3251.316} C_VEL
LIN {X 0,Y 447.612,Z 636.456,A -85,B 0,C 180,E1 3249.294,E2 3249.294} C_VEL
LIN {X 0,Y 446.93,Z 635.837,A -85,B 0,C 180,E1 3248.313,E2 3248.313} C_VEL
LIN {X 0,Y 445.785,Z 637.508,A -85,B 0,C 180,E1 3246.762,E2 3246.762} C_VEL
LIN {X 0,Y 444.909,Z 639.438,A -85,B 0,C 180,E1 3245.119,E2 3245.119} C_VEL
LIN {X 0,Y 444.811,Z 639.498,A -85,B 0,C 180,E1 3244.758,E2 3244.758} C_VEL
LIN {X 0,Y 444.867,Z 639.676,A -85,B 0,C 180,E1 3241.03,E2 3241.03} C_VEL
LIN {X 0,Y 446.425,Z 644.072,A -85,B 0,C 180,E1 3237.111,E2 3237.111} C_VEL
LIN {X 0,Y 447.398,Z 646.667,A -85,B 0,C 180,E1 3235.665,E2 3235.665} C_VEL
LIN {X 0,Y 427.945,Z 822.674,A -85,B 0,C 180,E1 3233.283,E2 3233.283} C_VEL
LIN {X 0,Y 423.767,Z 848.568,A -85,B 0,C 180,E1 3232.895,E2 3232.895} C_VEL
LIN {X 0,Y 417.388,Z 876.483,A -85,B 0,C 180,E1 3232.412,E2 3232.412} C_VEL
LIN {X 0,Y 411.398,Z 897.667,A -85,B 0,C 180,E1 3231.948,E2 3231.948} C_VEL
LIN {X 0,Y 404.511,Z 918.458,A -85,B 0,C 180,E1 3231.39,E2 3231.39} C_VEL
LIN {X 0,Y 396.491,Z 939.488,A -85,B 0,C 180,E1 3230.712,E2 3230.712} C_VEL
LIN {X 0,Y 385.508,Z 964.624,A -85,B 0,C 180,E1 3229.722,E2 3229.722} C_VEL
LIN {X 0,Y 374.288,Z 986.76,A -85,B 0,C 180,E1 3228.642,E2 3228.642} C_VEL
LIN {X 0,Y 363.546,Z 1005.875,A -85,B 0,C 180,E1 3227.522,E2 3227.522} C_VEL
LIN {X 0,Y 352.462,Z 1023.829,A -85,B 0,C 180,E1 3226.287,E2 3226.287} C_VEL
LIN {X 0,Y 339.913,Z 1042.456,A -85,B 0,C 180,E1 3224.762,E2 3224.762} C_VEL
LIN {X 0,Y 322.98,Z 1065.202,A -85,B 0,C 180,E1 3222.461,E2 3222.461} C_VEL
LIN {X 0,Y 309.027,Z 1082.242,A -85,B 0,C 180,E1 3220.315,E2 3220.315} C_VEL
LIN {X 0,Y 296.325,Z 1096.738,A -85,B 0,C 180,E1 3218.114,E2 3218.114} C_VEL
LIN {X 0,Y 283.328,Z 1110.682,A -85,B 0,C 180,E1 3215.575,E2 3215.575} C_VEL
LIN {X 0,Y 267.377,Z 1126.849,A -85,B 0,C 180,E1 3211.952,E2 3211.952} C_VEL
LIN {X 0,Y 251.891,Z 1141.396,A -85,B 0,C 180,E1 3207.727,E2 3207.727} C_VEL
LIN {X 0,Y 240.177,Z 1152.052,A -85,B 0,C 180,E1 3203.867,E2 3203.867} C_VEL
LIN {X 0,Y 228.969,Z 1162.033,A -85,B 0,C 180,E1 3199.408,E2 3199.408} C_VEL
LIN {X 0,Y 216.994,Z 1172.753,A -85,B 0,C 180,E1 3193.36,E2 3193.36} C_VEL
LIN {X 0,Y 206.943,Z 1181.845,A -85,B 0,C 180,E1 3186.463,E2 3186.463} C_VEL
LIN {X 0,Y 200.736,Z 1187.963,A -85,B 0,C 180,E1 3180.488,E2 3180.488} C_VEL
LIN {X 0,Y 196.54,Z 1192.667,A -85,B 0,C 180,E1 3174.657,E2 3174.657} C_VEL
LIN {X 0,Y 193.816,Z 1196.413,A -85,B 0,C 180,E1 3168.655,E2 3168.655} C_VEL
LIN {X 0,Y 192.438,Z 1199.071,A -85,B 0,C 180,E1 3162.911,E2 3162.911} C_VEL
LIN {X 0,Y 191.988,Z 1200.803,A -85,B 0,C 180,E1 3157.482,E2 3157.482} C_VEL
LIN {X 0,Y 191.916,Z 1201.781,A -85,B 0,C 180,E1 3152.091,E2 3152.091} C_VEL
LIN {X 0,Y 191.915,Z 1202.017,A -85,B 0,C 180,E1 3146.716,E2 3146.716} C_VEL
LIN {X 0,Y 192.08,Z 1201.38,A -85,B 0,C 180,E1 3140.715,E2 3140.715} C_VEL
LIN {X 0,Y 193.153,Z 1199.492,A -85,B 0,C 180,E1 3133.769,E2 3133.769} C_VEL
LIN {X 0,Y 195.685,Z 1196.587,A -85,B 0,C 180,E1 3127.151,E2 3127.151} C_VEL
LIN {X 0,Y 199.794,Z 1192.789,A -85,B 0,C 180,E1 3120.96,E2 3120.96} C_VEL
LIN {X 0,Y 205.662,Z 1187.963,A -85,B 0,C 180,E1 3114.994,E2 3114.994} C_VEL
LIN {X 0,Y 213.712,Z 1181.776,A -85,B 0,C 180,E1 3109.082,E2 3109.082} C_VEL
LIN {X 0,Y 226.122,Z 1172.615,A -85,B 0,C 180,E1 3102.402,E2 3102.402} C_VEL
LIN {X 0,Y 239.881,Z 1162.21,A -85,B 0,C 180,E1 3096.843,E2 3096.843} C_VEL
LIN {X 0,Y 252.89,Z 1152.159,A -85,B 0,C 180,E1 3092.633,E2 3092.633} C_VEL
LIN {X 0,Y 266.392,Z 1141.337,A -85,B 0,C 180,E1 3089.011,E2 3089.011} C_VEL
LIN {X 0,Y 283.057,Z 1127.31,A -85,B 0,C 180,E1 3085.273,E2 3085.273} C_VEL
LIN {X 0,Y 300.767,Z 1111.126,A -85,B 0,C 180,E1 3081.952,E2 3081.952} C_VEL
LIN {X 0,Y 315.266,Z 1096.933,A -85,B 0,C 180,E1 3079.622,E2 3079.622} C_VEL
LIN {X 0,Y 329.404,Z 1082.108,A -85,B 0,C 180,E1 3077.617,E2 3077.617} C_VEL
LIN {X 0,Y 343.049,Z 1066.716,A -85,B 0,C 180,E1 3075.882,E2 3075.882} C_VEL
LIN {X 0,Y 359.718,Z 1046.316,A -85,B 0,C 180,E1 3073.995,E2 3073.995} C_VEL
LIN {X 0,Y 375.296,Z 1024.825,A -85,B 0,C 180,E1 3072.409,E2 3072.409} C_VEL
LIN {X 0,Y 387.449,Z 1006.419,A -85,B 0,C 180,E1 3071.293,E2 3071.293} C_VEL
LIN {X 0,Y 398.431,Z 988.127,A -85,B 0,C 180,E1 3070.351,E2 3070.351} C_VEL
LIN {X 0,Y 409.525,Z 967.661,A -85,B 0,C 180,E1 3069.469,E2 3069.469} C_VEL
LIN {X 0,Y 422.12,Z 941.012,A -85,B 0,C 180,E1 3068.537,E2 3068.537} C_VEL
LIN {X 0,Y 431.051,Z 918.954,A -85,B 0,C 180,E1 3067.918,E2 3067.918} C_VEL
LIN {X 0,Y 438.297,Z 898.314,A -85,B 0,C 180,E1 3067.44,E2 3067.44} C_VEL
LIN {X 0,Y 444.726,Z 876.838,A -85,B 0,C 180,E1 3067.035,E2 3067.035} C_VEL
LIN {X 0,Y 451.302,Z 849.961,A -85,B 0,C 180,E1 3066.627,E2 3066.627} C_VEL
LIN {X 0,Y 456.045,Z 822.566,A -85,B 0,C 180,E1 3066.256,E2 3066.256} C_VEL
LIN {X 0,Y 473.284,Z 679.56,A -85,B 0,C 180,E1 3064.434,E2 3064.434} C_VEL
LIN {X 0,Y 474.46,Z 669.744,A -85,B 0,C 180,E1 3064.291,E2 3064.291} C_VEL
LIN {X 0,Y 474.455,Z 668.6,A -85,B 0,C 180,E1 3062.778,E2 3062.778} C_VEL
LIN {X 0,Y 474.437,Z 669.902,A -85,B 0,C 180,E1 3061.525,E2 3061.525} C_VEL
LIN {X 0,Y 456.124,Z 821.756,A -85,B 0,C 180,E1 3059.592,E2 3059.592} C_VEL
LIN {X 0,Y 451.547,Z 848.297,A -85,B 0,C 180,E1 3059.234,E2 3059.234} C_VEL
LIN {X 0,Y 444.973,Z 875.47,A -85,B 0,C 180,E1 3058.808,E2 3058.808} C_VEL
LIN {X 0,Y 438.615,Z 896.823,A -85,B 0,C 180,E1 3058.384,E2 3058.384} C_VEL
LIN {X 0,Y 431.483,Z 917.235,A -85,B 0,C 180,E1 3057.893,E2 3057.893} C_VEL
LIN {X 0,Y 423.089,Z 938.096,A -85,B 0,C 180,E1 3057.291,E2 3057.291} C_VEL
LIN {X 0,Y 411.745,Z 962.717,A -85,B 0,C 180,E1 3056.426,E2 3056.426} C_VEL
LIN {X 0,Y 399.222,Z 985.954,A -85,B 0,C 180,E1 3055.416,E2 3055.416} C_VEL
LIN {X 0,Y 388.263,Z 1004.25,A -85,B 0,C 180,E1 3054.457,E2 3054.457} C_VEL
LIN {X 0,Y 376.471,Z 1022.135,A -85,B 0,C 180,E1 3053.364,E2 3053.364} C_VEL
LIN {X 0,Y 362.989,Z 1040.805,A -85,B 0,C 180,E1 3051.993,E2 3051.993} C_VEL
LIN {X 0,Y 345.213,Z 1062.957,A -85,B 0,C 180,E1 3049.985,E2 3049.985} C_VEL
LIN {X 0,Y 330.096,Z 1079.974,A -85,B 0,C 180,E1 3048.061,E2 3048.061} C_VEL
LIN {X 0,Y 316.349,Z 1094.323,A -85,B 0,C 180,E1 3046.101,E2 3046.101} C_VEL
LIN {X 0,Y 301.962,Z 1108.326,A -85,B 0,C 180,E1 3043.791,E2 3043.791} C_VEL
LIN {X 0,Y 284.229,Z 1124.448,A -85,B 0,C 180,E1 3040.476,E2 3040.476} C_VEL
LIN {X 0,Y 267.636,Z 1138.258,A -85,B 0,C 180,E1 3036.784,E2 3036.784} C_VEL
LIN {X 0,Y 254.234,Z 1148.869,A -85,B 0,C 180,E1 3033.221,E2 3033.221} C_VEL
LIN {X 0,Y 241.86,Z 1158.268,A -85,B 0,C 180,E1 3029.303,E2 3029.303} C_VEL
LIN {X 0,Y 229.54,Z 1167.351,A -85,B 0,C 180,E1 3024.543,E2 3024.543} C_VEL
LIN {X 0,Y 216.096,Z 1177.143,A -85,B 0,C 180,E1 3017.757,E2 3017.757} C_VEL
LIN {X 0,Y 206.965,Z 1183.826,A -85,B 0,C 180,E1 3011.441,E2 3011.441} C_VEL
LIN {X 0,Y 200.621,Z 1188.758,A -85,B 0,C 180,E1 3005.318,E2 3005.318} C_VEL
LIN {X 0,Y 196.168,Z 1192.592,A -85,B 0,C 180,E1 2998.96,E2 2998.96} C_VEL
LIN {X 0,Y 193.567,Z 1195.247,A -85,B 0,C 180,E1 2992.792,E2 2992.792} C_VEL
LIN {X 0,Y 192.361,Z 1196.89,A -85,B 0,C 180,E1 2986.922,E2 2986.922} C_VEL
LIN {X 0,Y 191.977,Z 1197.658,A -85,B 0,C 180,E1 2981.711,E2 2981.711} C_VEL
LIN {X 0,Y 191.913,Z 1197.791,A -85,B 0,C 180,E1 2976.581,E2 2976.581} C_VEL
LIN {X 0,Y 191.955,Z 1197.166,A -85,B 0,C 180,E1 2970.894,E2 2970.894} C_VEL
LIN {X 0,Y 192.352,Z 1195.526,A -85,B 0,C 180,E1 2964.63,E2 2964.63} C_VEL
